KUKA KRL program: MyProgram_336().src

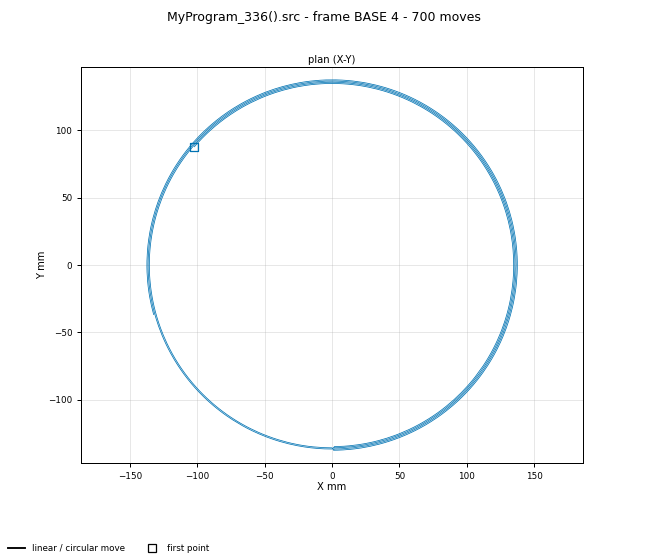
[picture p0: tool path of MyProgram_336().src in frame BASE 4, 700 of 700 moves have a stored position in this frame; points joined in program order, loops and branches not executed]
&ACCESS RVP
&REL 1
&PARAM TEMPLATE = C:\KRC\Roboter\Template\vorgabe
&PARAM EDITMASK = *
DEF MyProgram_336()
; ---- Setting reference (Base) ----
$BASE = BASE_DATA[4]

; --------------------------
; ---- Setting tool (TCP) ----
$TOOL = TOOL_DATA[3]
; --------------------------

$VEL.CP = VEL_APROX_PRINT
Startdeposition()
$VEL.CP = VEL_PRINT
LIN {X -102.3113,Y 87.8805,Z 190,A 136.75,B 1.0314,C -0.0375,E1 0.9175,E2 317.7495} C_DIS
LIN {X -99.637,Y 90.9019,Z 190,A 134.8768,B 1.0314,C -0.0407,E1 0.9211,E2 319.6393} C_DIS
LIN {X -96.5901,Y 94.1334,Z 190,A 132.7694,B 1.0312,C -0.0441,E1 0.9252,E2 321.7696} C_DIS
LIN {X -92.9272,Y 97.7507,Z 190,A 130.473,B 1.031,C -0.0478,E1 0.9299,E2 324.0767} C_DIS
LIN {X -90.6554,Y 99.8606,Z 190,A 129.0008,B 1.031,C -0.0499,E1 0.933,E2 325.565} C_DIS
LIN {X -87.4566,Y 102.6738,Z 190,A 127.0141,B 1.0308,C -0.0527,E1 0.9372,E2 327.5698} C_DIS
LIN {X -83.8464,Y 105.6426,Z 190,A 124.8651,B 1.0306,C -0.0556,E1 0.942,E2 329.7352} C_DIS
LIN {X -79.6041,Y 108.8753,Z 190,A 122.7567,B 1.0305,C -0.0588,E1 0.9467,E2 331.8252} C_DIS
LIN {X -75.5574,Y 111.7212,Z 190,A 120.2221,B 1.0303,C -0.0612,E1 0.9527,E2 334.4052} C_DIS
LIN {X -71.0559,Y 114.6372,Z 190,A 118.0805,B 1.0301,C -0.064,E1 0.9577,E2 336.5308} C_DIS
LIN {X -66.7987,Y 117.1687,Z 190,A 115.5078,B 1.0301,C -0.0659,E1 0.9641,E2 339.1524} C_DIS
LIN {X -63.7892,Y 118.8339,Z 190,A 114.076,B 1.0299,C -0.0674,E1 0.9676,E2 340.5803} C_DIS
LIN {X -60.168,Y 120.7068,Z 190,A 112.074,B 1.0299,C -0.0687,E1 0.9727,E2 342.61} C_DIS
LIN {X -55.6939,Y 122.8359,Z 190,A 110.1767,B 1.0297,C -0.0706,E1 0.9775,E2 344.4841} C_DIS
LIN {X -53.3762,Y 123.8589,Z 190,A 108.9368,B 1.0297,C -0.0712,E1 0.9808,E2 345.7408} C_DIS
LIN {X -50.0858,Y 125.2261,Z 190,A 107.31,B 1.0297,C -0.0721,E1 0.9851,E2 347.3788} C_DIS
LIN {X -46.763,Y 126.5053,Z 190,A 105.8623,B 1.0295,C -0.073,E1 0.9889,E2 348.8188} C_DIS
LIN {X -42.2008,Y 128.0989,Z 190,A 103.8391,B 1.0295,C -0.0741,E1 0.9943,E2 350.8378} C_DIS
LIN {X -39.3457,Y 129.0038,Z 190,A 102.4581,B 1.0295,C -0.0745,E1 0.998,E2 352.2297} C_DIS
LIN {X -36.135,Y 129.9398,Z 190,A 100.9752,B 1.0295,C -0.0749,E1 1.0021,E2 353.7185} C_DIS
LIN {X -32.8396,Y 130.8119,Z 190,A 99.599,B 1.0294,C -0.0754,E1 1.0058,E2 355.0863} C_DIS
LIN {X -29.9981,Y 131.4922,Z 190,A 98.2261,B 1.0294,C -0.0754,E1 1.0096,E2 356.4725} C_DIS
LIN {X -26.2178,Y 132.2996,Z 190,A 96.5812,B 1.0294,C -0.0757,E1 1.0142,E2 358.1171} C_DIS
LIN {X -20.3497,Y 133.327,Z 190,A 94.0999,B 1.0294,C -0.0759,E1 1.0211,E2 360.5919} C_DIS
LIN {X -16.2447,Y 133.8892,Z 190,A 92.3486,B 1.0294,C -0.0759,E1 1.026,E2 362.3415} C_DIS
LIN {X -12.8323,Y 134.259,Z 190,A 90.8849,B 1.0294,C -0.0756,E1 1.0301,E2 363.8052} C_DIS
LIN {X -8.2772,Y 134.6166,Z 190,A 89.0248,B 1.0294,C -0.0753,E1 1.0353,E2 365.6559} C_DIS
LIN {X -4.9946,Y 134.7786,Z 190,A 87.4221,B 1.0294,C -0.0744,E1 1.0399,E2 367.2799} C_DIS
LIN {X -0.1697,Y 134.872,Z 190,A 85.4609,B 1.0294,C -0.0738,E1 1.0454,E2 369.2309} C_DIS
LIN {X 3.9569,Y 134.813,Z 190,A 83.7686,B 1.0295,C -0.0731,E1 1.0502,E2 370.9162} C_DIS
LIN {X 8.1399,Y 134.6251,Z 190,A 82.1087,B 1.0295,C -0.0724,E1 1.0548,E2 372.5628} C_DIS
LIN {X 11.7899,Y 134.3552,Z 190,A 80.705,B 1.0296,C -0.0718,E1 1.0587,E2 373.95} C_DIS
LIN {X 15.0526,Y 134.0296,Z 190,A 79.3206,B 1.0296,C -0.0708,E1 1.0626,E2 375.333} C_DIS
LIN {X 18.9857,Y 133.5278,Z 190,A 77.6744,B 1.0298,C -0.0696,E1 1.0672,E2 376.9746} C_DIS
LIN {X 22.5244,Y 132.9769,Z 190,A 76.1298,B 1.0298,C -0.0683,E1 1.0715,E2 378.5212} C_DIS
LIN {X 26.8707,Y 132.1668,Z 190,A 74.3853,B 1.03,C -0.0669,E1 1.0763,E2 380.2509} C_DIS
LIN {X 30.9711,Y 131.268,Z 190,A 72.7965,B 1.03,C -0.0657,E1 1.0806,E2 381.8185} C_DIS
LIN {X 33.4746,Y 130.6507,Z 190,A 71.6675,B 1.0301,C -0.0645,E1 1.0837,E2 382.9507} C_DIS
LIN {X 37.5809,Y 129.5293,Z 190,A 69.9323,B 1.0302,C -0.0626,E1 1.0884,E2 384.6777} C_DIS
LIN {X 41.1171,Y 128.4501,Z 190,A 68.1111,B 1.0304,C -0.0599,E1 1.0934,E2 386.5253} C_DIS
LIN {X 44.8572,Y 127.1943,Z 190,A 66.979,B 1.0304,C -0.0596,E1 1.0963,E2 387.5987} C_DIS
LIN {X 49.4196,Y 125.4914,Z 190,A 64.9699,B 1.0306,C -0.057,E1 1.1015,E2 389.6009} C_DIS
LIN {X 52.5027,Y 124.2329,Z 190,A 63.4716,B 1.0306,C -0.0547,E1 1.1055,E2 391.108} C_DIS
LIN {X 56.3475,Y 122.5359,Z 190,A 61.913,B 1.0308,C -0.0529,E1 1.1094,E2 392.6417} C_DIS
LIN {X 59.8944,Y 120.8418,Z 190,A 60.3889,B 1.0308,C -0.0508,E1 1.1132,E2 394.1497} C_DIS
LIN {X 65.5035,Y 117.8978,Z 190,A 58.0418,B 1.031,C -0.0478,E1 1.119,E2 396.4588} C_DIS
LIN {X 68.3222,Y 116.2869,Z 190,A 56.6628,B 1.0311,C -0.0454,E1 1.1223,E2 397.8377} C_DIS
LIN {X 71.8669,Y 114.1303,Z 190,A 54.9703,B 1.0313,C -0.0426,E1 1.1263,E2 399.5224} C_DIS
LIN {X 74.5809,Y 112.376,Z 190,A 53.7411,B 1.0313,C -0.0407,E1 1.1292,E2 400.7356} C_DIS
LIN {X 78.1084,Y 109.9537,Z 190,A 52.01,B 1.0314,C -0.0377,E1 1.1332,E2 402.4571} C_DIS
LIN {X 81.7669,Y 107.2603,Z 190,A 50.3364,B 1.0315,C -0.035,E1 1.1369,E2 404.102} C_DIS
LIN {X 84.8066,Y 104.8734,Z 190,A 48.8019,B 1.0316,C -0.0322,E1 1.1402,E2 405.6245} C_DIS
LIN {X 88.0931,Y 102.1282,Z 190,A 47.1444,B 1.0317,C -0.0292,E1 1.1437,E2 407.264} C_DIS
LIN {X 91.5195,Y 99.0698,Z 190,A 45.3771,B 1.0318,C -0.0259,E1 1.1473,E2 409.0107} C_DIS
LIN {X 93.7332,Y 96.9776,Z 190,A 44.1924,B 1.0318,C -0.0236,E1 1.1497,E2 410.1831} C_DIS
LIN {X 96.9928,Y 93.7175,Z 190,A 42.4386,B 1.0319,C -0.0203,E1 1.1531,E2 411.9139} C_DIS
LIN {X 99.9264,Y 90.583,Z 190,A 40.7946,B 1.0319,C -0.017,E1 1.1562,E2 413.5376} C_DIS
LIN {X 102.9019,Y 87.1883,Z 190,A 39.069,B 1.032,C -0.0135,E1 1.1593,E2 415.2415} C_DIS
LIN {X 105.5381,Y 83.9777,Z 190,A 37.4765,B 1.032,C -0.0102,E1 1.1621,E2 416.8145} C_DIS
LIN {X 108.1139,Y 80.6346,Z 190,A 36.0003,B 1.0321,C -0.0075,E1 1.1646,E2 418.2544} C_DIS
LIN {X 110.3862,Y 77.4954,Z 190,A 34.2134,B 1.0321,C -0.0029,E1 1.1675,E2 420.0579} C_DIS
LIN {X 112.2299,Y 74.7998,Z 190,A 33.1847,B 1.0321,C -0.0012,E1 1.169,E2 421.0454} C_DIS
LIN {X 114.6113,Y 71.0975,Z 190,A 31.5626,B 1.0321,C 0.0022,E1 1.1714,E2 422.6389} C_DIS
LIN {X 116.9008,Y 67.2672,Z 190,A 29.7748,B 1.0321,C 0.0065,E1 1.1739,E2 424.4146} C_DIS
LIN {X 118.7485,Y 63.9481,Z 190,A 28.4203,B 1.0321,C 0.0093,E1 1.1757,E2 425.739} C_DIS
LIN {X 120.388,Y 60.8022,Z 190,A 27.1011,B 1.0321,C 0.0122,E1 1.1774,E2 427.0364} C_DIS
LIN {X 122.4869,Y 56.4534,Z 190,A 25.2811,B 1.0321,C 0.0164,E1 1.1795,E2 428.8296} C_DIS
LIN {X 124.0395,Y 52.9585,Z 190,A 23.9004,B 1.0319,C 0.0194,E1 1.181,E2 430.1818} C_DIS
LIN {X 125.287,Y 49.9347,Z 190,A 22.621,B 1.0319,C 0.0225,E1 1.1824,E2 431.4484} C_DIS
LIN {X 126.9081,Y 45.6549,Z 190,A 20.9084,B 1.0318,C 0.0265,E1 1.184,E2 433.1339} C_DIS
LIN {X 127.9726,Y 42.58,Z 190,A 19.6934,B 1.0318,C 0.0294,E1 1.1851,E2 434.3292} C_DIS
LIN {X 129.125,Y 38.9496,Z 190,A 18.2521,B 1.0316,C 0.0328,E1 1.1863,E2 435.7498} C_DIS
LIN {X 130.0995,Y 35.5641,Z 190,A 16.9404,B 1.0316,C 0.0359,E1 1.1872,E2 437.0398} C_DIS
LIN {X 130.8248,Y 32.7889,Z 190,A 15.8845,B 1.0314,C 0.0384,E1 1.188,E2 438.0763} C_DIS
LIN {X 131.5462,Y 29.7614,Z 190,A 14.7035,B 1.0314,C 0.0413,E1 1.1887,E2 439.2406} C_DIS
LIN {X 132.2329,Y 26.5457,Z 190,A 13.4674,B 1.0312,C 0.0443,E1 1.1894,E2 440.4576} C_DIS
LIN {X 132.8388,Y 23.327,Z 190,A 12.2792,B 1.0311,C 0.0471,E1 1.19,E2 441.6216} C_DIS
LIN {X 133.4079,Y 19.8242,Z 190,A 10.9318,B 1.0309,C 0.0504,E1 1.1905,E2 442.95} C_DIS
LIN {X 133.8223,Y 16.7998,Z 190,A 9.5869,B 1.0307,C 0.0543,E1 1.191,E2 444.3014} C_DIS
LIN {X 134.3804,Y 11.4921,Z 190,A 7.7327,B 1.0305,C 0.0584,E1 1.1915,E2 446.1055} C_DIS
LIN {X 134.6681,Y 7.4209,Z 190,A 6.3001,B 1.0303,C 0.0616,E1 1.1918,E2 447.5015} C_DIS
LIN {X 134.7793,Y 4.9766,Z 190,A 5.324,B 1.0301,C 0.0642,E1 1.1918,E2 448.4702} C_DIS
LIN {X 134.8718,Y 0.2243,Z 190,A 3.6075,B 1.0299,C 0.0682,E1 1.1919,E2 450.1498} C_DIS
LIN {X 134.8428,Y -2.814,Z 190,A 2.2229,B 1.0296,C 0.0723,E1 1.1919,E2 451.5469} C_DIS
LIN {X 134.6641,Y -7.5005,Z 190,A 0.6838,B 1.0294,C 0.0754,E1 1.1917,E2 453.03} C_DIS
LIN {X 134.3382,Y -11.9912,Z 190,A -1.3076,B 1.0289,C 0.0812,E1 1.1912,E2 455.0324} C_DIS
LIN {X 133.9962,Y -15.3478,Z 190,A -2.2241,B 1.0289,C 0.0824,E1 1.191,E2 455.8842} C_DIS
LIN {X 133.6072,Y -18.4298,Z 190,A -3.5585,B 1.0285,C 0.0861,E1 1.1905,E2 457.2212} C_DIS
LIN {X 132.9067,Y -22.945,Z 190,A -5.1491,B 1.0282,C 0.0896,E1 1.1898,E2 458.7683} C_DIS
LIN {X 132.425,Y -25.5689,Z 190,A -6.1171,B 1.028,C 0.0918,E1 1.1893,E2 459.7157} C_DIS
LIN {X 131.6541,Y -29.2892,Z 190,A -7.6683,B 1.0277,C 0.0959,E1 1.1884,E2 461.2599} C_DIS
LIN {X 130.7208,Y -33.1985,Z 190,A -9.1638,B 1.0273,C 0.0995,E1 1.1874,E2 462.7291} C_DIS
LIN {X 129.6374,Y -37.2116,Z 190,A -11.2094,B 1.0267,C 0.1058,E1 1.1858,E2 464.812} C_DIS
LIN {X 128.1582,Y -42.0227,Z 190,A -12.4751,B 1.0266,C 0.1069,E1 1.1848,E2 465.966} C_DIS
LIN {X 127.2027,Y -44.833,Z 190,A -13.6596,B 1.0263,C 0.1098,E1 1.1838,E2 467.1414} C_DIS
LIN {X 126.0621,Y -47.9462,Z 190,A -14.8848,B 1.026,C 0.1126,E1 1.1826,E2 468.3436} C_DIS
LIN {X 124.9341,Y -50.81,Z 190,A -16.3072,B 1.0255,C 0.1166,E1 1.1811,E2 469.7819} C_DIS
LIN {X 122.8544,Y -55.6527,Z 190,A -18.0514,B 1.0251,C 0.1199,E1 1.1792,E2 471.4627} C_DIS
LIN {X 121.7034,Y -58.1231,Z 190,A -19.1462,B 1.0248,C 0.1225,E1 1.1779,E2 472.5499} C_DIS
LIN {X 119.7934,Y -61.9695,Z 190,A -20.702,B 1.0244,C 0.1258,E1 1.176,E2 474.0716} C_DIS
LIN {X 118.0054,Y -65.3091,Z 190,A -22.1982,B 1.024,C 0.1293,E1 1.174,E2 475.5539} C_DIS
LIN {X 115.8653,Y -69.0347,Z 190,A -23.7083,B 1.0236,C 0.1322,E1 1.1719,E2 477.0234} C_DIS
LIN {X 113.9593,Y -72.1378,Z 190,A -25.1095,B 1.0232,C 0.1353,E1 1.1699,E2 478.4062} C_DIS
LIN {X 112.1061,Y -74.9853,Z 190,A -26.594,B 1.0227,C 0.139,E1 1.1676,E2 479.8974} C_DIS
LIN {X 106.1881,Y -83.1545,Z 190,A -30.2178,B 1.0218,C 0.1459,E1 1.1617,E2 483.4355} C_DIS
LIN {X 104.0205,Y -85.8506,Z 190,A -32.1493,B 1.0209,C 0.1516,E1 1.1582,E2 485.4304} C_DIS
LIN {X 100.756,Y -89.6603,Z 190,A -33.3836,B 1.0209,C 0.1519,E1 1.1561,E2 486.5452} C_DIS
LIN {X 95.9069,Y -94.8289,Z 190,A -36.3467,B 1.0199,C 0.1583,E1 1.1504,E2 489.5043} C_DIS
LIN {X 90.6268,Y -99.8866,Z 190,A -38.942,B 1.0193,C 0.1624,E1 1.1452,E2 492.0322} C_DIS
LIN {X 84.6508,Y -104.999,Z 190,A -42.6037,B 1.0179,C 0.1707,E1 1.1373,E2 495.7404} C_DIS
LIN {X 80.9291,Y -107.894,Z 190,A -43.8915,B 1.0179,C 0.1712,E1 1.1346,E2 496.9318} C_DIS
LIN {X 78.2121,Y -109.8795,Z 190,A -45.324,B 1.0174,C 0.1739,E1 1.1313,E2 498.3657} C_DIS
LIN {X 74.889,Y -112.1704,Z 190,A -46.9282,B 1.0169,C 0.1766,E1 1.1276,E2 499.956} C_DIS
LIN {X 71.4377,Y -114.3995,Z 190,A -48.5106,B 1.0165,C 0.1789,E1 1.1239,E2 501.5172} C_DIS
LIN {X 66.7848,Y -117.1765,Z 190,A -50.4352,B 1.0161,C 0.1812,E1 1.1194,E2 503.3913} C_DIS
LIN {X 64.1989,Y -118.6138,Z 190,A -51.8491,B 1.0156,C 0.1839,E1 1.1158,E2 504.8279} C_DIS
LIN {X 60.9277,Y -120.3242,Z 190,A -53.1719,B 1.0154,C 0.1854,E1 1.1126,E2 506.1177} C_DIS
LIN {X 57.1495,Y -122.1651,Z 190,A -54.7355,B 1.015,C 0.1872,E1 1.1087,E2 507.6517} C_DIS
LIN {X 50.0805,Y -125.2282,Z 190,A -57.8745,B 1.0142,C 0.1913,E1 1.1006,E2 510.7745} C_DIS
LIN {X 46.6988,Y -126.5294,Z 190,A -59.694,B 1.0136,C 0.1945,E1 1.0957,E2 512.6342} C_DIS
LIN {X 43.1235,Y -127.7916,Z 190,A -60.7374,B 1.0136,C 0.1943,E1 1.0931,E2 513.5994} C_DIS
LIN {X 40.4042,Y -128.6779,Z 190,A -61.97,B 1.0134,C 0.1958,E1 1.0898,E2 514.8354} C_DIS
LIN {X 37.734,Y -129.4845,Z 190,A -63.1158,B 1.0131,C 0.1971,E1 1.0867,E2 515.9765} C_DIS
LIN {X 34.6217,Y -130.3511,Z 190,A -64.3488,B 1.013,C 0.1981,E1 1.0834,E2 517.1907} C_DIS
LIN {X 31.3438,Y -131.1782,Z 190,A -65.8293,B 1.0126,C 0.1997,E1 1.0793,E2 518.6785} C_DIS
LIN {X 27.9921,Y -131.9347,Z 190,A -67.1371,B 1.0124,C 0.2006,E1 1.0758,E2 519.9659} C_DIS
LIN {X 24.3157,Y -132.6618,Z 190,A -68.7166,B 1.0122,C 0.2021,E1 1.0714,E2 521.5447} C_DIS
LIN {X 19.7753,Y -133.4139,Z 190,A -71.0449,B 1.0116,C 0.205,E1 1.0648,E2 523.9265} C_DIS
LIN {X 15.397,Y -133.9903,Z 190,A -72.2873,B 1.0117,C 0.2043,E1 1.0615,E2 525.0811} C_DIS
LIN {X 12.6782,Y -134.2738,Z 190,A -73.5571,B 1.0115,C 0.2054,E1 1.0579,E2 526.3668} C_DIS
LIN {X 8.7907,Y -134.585,Z 190,A -75.5639,B 1.011,C 0.2076,E1 1.0521,E2 528.4237} C_DIS
LIN {X 4.4935,Y -134.7977,Z 190,A -76.8327,B 1.0112,C 0.2068,E1 1.0488,E2 529.615} C_DIS
LIN {X 1.7112,Y -134.8611,Z 190,A -78.397,B 1.0108,C 0.2085,E1 1.0442,E2 531.2338} C_DIS
LIN {X 1.7112,Y -134.8611,Z 190,A -78.397,B 1.0108,C 0.2085,E1 1.0442,E2 531.2338} C_DIS
Enddeposition()
LIN {X 0.9737,Y -135.7663,Z 190,A -78.1161,B 1.011,C 0.2073,E1 1.045,E2 530.8941} C_DIS
Startdeposition()
$VEL.CP = VEL_PRINT
LIN {X 6.9745,Y -135.5906,Z 190,A -75.108,B 1.0116,C 0.2046,E1 1.0537,E2 527.8168} C_DIS
LIN {X 15.8798,Y -134.8379,Z 190,A -71.5086,B 1.012,C 0.2026,E1 1.0638,E2 524.2401} C_DIS
LIN {X 22.5103,Y -133.8906,Z 190,A -68.8862,B 1.0123,C 0.2009,E1 1.071,E2 521.6453} C_DIS
LIN {X 25.8344,Y -133.2894,Z 190,A -67.4107,B 1.0126,C 0.1994,E1 1.0751,E2 520.1618} C_DIS
LIN {X 28.9884,Y -132.6392,Z 190,A -66.1615,B 1.0128,C 0.1985,E1 1.0785,E2 518.9274} C_DIS
LIN {X 33.1343,Y -131.6645,Z 190,A -64.4396,B 1.0131,C 0.1969,E1 1.0832,E2 517.2151} C_DIS
LIN {X 36.5609,Y -130.7541,Z 190,A -63.091,B 1.0133,C 0.1958,E1 1.0869,E2 515.8865} C_DIS
LIN {X 39.6778,Y -129.8422,Z 190,A -61.7393,B 1.0136,C 0.1943,E1 1.0905,E2 514.5366} C_DIS
LIN {X 42.6723,Y -128.8893,Z 190,A -60.4442,B 1.0139,C 0.1928,E1 1.094,E2 513.245} C_DIS
LIN {X 47.1805,Y -127.3088,Z 190,A -58.7448,B 1.0141,C 0.1914,E1 1.0984,E2 511.5893} C_DIS
LIN {X 49.6539,Y -126.3647,Z 190,A -56.71,B 1.0151,C 0.1861,E1 1.1041,E2 509.4227} C_DIS
LIN {X 55.9848,Y -123.6906,Z 190,A -54.8821,B 1.0151,C 0.1864,E1 1.1084,E2 507.7458} C_DIS
LIN {X 59.6108,Y -121.984,Z 190,A -53.2483,B 1.0155,C 0.184,E1 1.1125,E2 506.1189} C_DIS
LIN {X 62.986,Y -120.2749,Z 190,A -51.8669,B 1.0158,C 0.1824,E1 1.1159,E2 504.7667} C_DIS
LIN {X 66.363,Y -118.4475,Z 190,A -49.6176,B 1.0167,C 0.177,E1 1.1216,E2 502.4272} C_DIS
LIN {X 71.4623,Y -115.4429,Z 190,A -47.9158,B 1.0169,C 0.1762,E1 1.1254,E2 500.8363} C_DIS
LIN {X 74.8801,Y -113.2558,Z 190,A -46.4071,B 1.0173,C 0.1741,E1 1.1289,E2 499.3549} C_DIS
LIN {X 77.3617,Y -111.5753,Z 190,A -45.1498,B 1.0176,C 0.1718,E1 1.1318,E2 498.0977} C_DIS
LIN {X 82.7712,Y -107.6238,Z 190,A -42.5903,B 1.0183,C 0.1676,E1 1.1375,E2 495.5736} C_DIS
LIN {X 86.0264,Y -105.0396,Z 190,A -40.5384,B 1.0191,C 0.1627,E1 1.1421,E2 493.4787} C_DIS
LIN {X 89.8971,Y -101.7465,Z 190,A -38.9851,B 1.0194,C 0.1611,E1 1.1452,E2 492.0065} C_DIS
LIN {X 93.6072,Y -98.3443,Z 190,A -37.1127,B 1.0199,C 0.1579,E1 1.149,E2 490.1675} C_DIS
LIN {X 96.9051,Y -95.0959,Z 190,A -34.9295,B 1.0207,C 0.1525,E1 1.1533,E2 487.9509} C_DIS
LIN {X 100.2823,Y -91.5282,Z 190,A -33.4715,B 1.0209,C 0.151,E1 1.1559,E2 486.5768} C_DIS
LIN {X 104.4413,Y -86.7519,Z 190,A -31.0792,B 1.0216,C 0.1463,E1 1.1602,E2 484.2211} C_DIS
LIN {X 109.0323,Y -80.9064,Z 190,A -28.199,B 1.0225,C 0.1403,E1 1.1651,E2 481.3739} C_DIS
LIN {X 113.3577,Y -74.7254,Z 190,A -25.4327,B 1.0232,C 0.1347,E1 1.1694,E2 478.6624} C_DIS
LIN {X 115.8481,Y -70.8032,Z 190,A -23.9195,B 1.0235,C 0.1322,E1 1.1716,E2 477.2086} C_DIS
LIN {X 117.5871,Y -67.8759,Z 190,A -22.4205,B 1.024,C 0.1283,E1 1.1737,E2 475.7001} C_DIS
LIN {X 119.8326,Y -63.8285,Z 190,A -20.645,B 1.0245,C 0.1243,E1 1.176,E2 473.9472} C_DIS
LIN {X 121.6063,Y -60.3763,Z 190,A -19.3533,B 1.0248,C 0.1219,E1 1.1776,E2 472.7009} C_DIS
LIN {X 123.017,Y -57.4489,Z 190,A -18.0289,B 1.0252,C 0.1186,E1 1.1792,E2 471.3818} C_DIS
LIN {X 124.5269,Y -54.0963,Z 190,A -16.0232,B 1.0259,C 0.1121,E1 1.1815,E2 469.3139} C_DIS
LIN {X 126.7317,Y -48.7098,Z 190,A -14.4966,B 1.0261,C 0.1106,E1 1.1829,E2 467.9106} C_DIS
LIN {X 129.6888,Y -40.179,Z 190,A -11.0276,B 1.027,C 0.1023,E1 1.186,E2 464.4846} C_DIS
LIN {X 130.8301,Y -36.2891,Z 190,A -9.5625,B 1.0273,C 0.0989,E1 1.1871,E2 463.0508} C_DIS
LIN {X 131.8524,Y -32.3826,Z 190,A -8.0428,B 1.0276,C 0.0953,E1 1.1881,E2 461.5544} C_DIS
LIN {X 132.804,Y -28.225,Z 190,A -6.4515,B 1.028,C 0.0915,E1 1.1891,E2 459.9894} C_DIS
LIN {X 133.632,Y -23.9971,Z 190,A -4.9377,B 1.0283,C 0.0881,E1 1.1898,E2 458.5143} C_DIS
LIN {X 134.1433,Y -20.952,Z 190,A -3.7879,B 1.0285,C 0.0854,E1 1.1903,E2 457.3836} C_DIS
LIN {X 134.6414,Y -17.4673,Z 190,A -1.6977,B 1.0291,C 0.0779,E1 1.1911,E2 455.2133} C_DIS
LIN {X 135.3223,Y -11.0204,Z 190,A 0.051,B 1.0293,C 0.0757,E1 1.1915,E2 453.5921} C_DIS
LIN {X 135.5533,Y -7.6919,Z 190,A 1.7384,B 1.0296,C 0.0703,E1 1.1918,E2 451.8677} C_DIS
LIN {X 135.745,Y -2.6227,Z 190,A 3.0238,B 1.0297,C 0.0689,E1 1.1918,E2 450.6915} C_DIS
LIN {X 135.7107,Y 4.0127,Z 190,A 5.6323,B 1.0302,C 0.0622,E1 1.1918,E2 448.1062} C_DIS
LIN {X 135.4983,Y 8.5847,Z 190,A 7.7512,B 1.0305,C 0.0557,E1 1.1914,E2 445.9623} C_DIS
LIN {X 135.0989,Y 13.4892,Z 190,A 9.3749,B 1.0307,C 0.0524,E1 1.191,E2 444.3954} C_DIS
LIN {X 134.6912,Y 17.0876,Z 190,A 10.5353,B 1.0308,C 0.0501,E1 1.1906,E2 443.2809} C_DIS
LIN {X 134.0881,Y 21.3087,Z 190,A 11.9098,B 1.0309,C 0.0474,E1 1.19,E2 441.9589} C_DIS
LIN {X 133.4862,Y 24.805,Z 190,A 13.3118,B 1.0311,C 0.0438,E1 1.1893,E2 440.5682} C_DIS
LIN {X 132.8466,Y 28.0274,Z 190,A 14.6057,B 1.0312,C 0.0405,E1 1.1886,E2 439.2852} C_DIS
LIN {X 131.9947,Y 31.7922,Z 190,A 15.9489,B 1.0314,C 0.0375,E1 1.1878,E2 437.9768} C_DIS
LIN {X 131.3208,Y 34.4742,Z 190,A 17.0801,B 1.0314,C 0.0345,E1 1.187,E2 436.8497} C_DIS
LIN {X 130.3166,Y 38.0909,Z 190,A 18.4506,B 1.0316,C 0.0313,E1 1.186,E2 435.5049} C_DIS
LIN {X 129.0944,Y 42.0543,Z 190,A 20.0951,B 1.0316,C 0.0272,E1 1.1846,E2 433.8729} C_DIS
LIN {X 127.6763,Y 46.1746,Z 190,A 22.1395,B 1.0318,C 0.0212,E1 1.1826,E2 431.8025} C_DIS
LIN {X 125.8411,Y 50.9644,Z 190,A 23.4871,B 1.0318,C 0.0197,E1 1.1813,E2 430.5545} C_DIS
LIN {X 124.4351,Y 54.3084,Z 190,A 25.3938,B 1.0319,C 0.0137,E1 1.1792,E2 428.6014} C_DIS
LIN {X 122.3616,Y 58.8305,Z 190,A 26.73,B 1.0319,C 0.0121,E1 1.1777,E2 427.3577} C_DIS
LIN {X 120.5356,Y 62.4896,Z 190,A 28.2924,B 1.0319,C 0.0085,E1 1.1757,E2 425.8145} C_DIS
LIN {X 118.5328,Y 66.2113,Z 190,A 29.8531,B 1.032,C 0.0051,E1 1.1736,E2 424.2802} C_DIS
LIN {X 115.3809,Y 71.5621,Z 190,A 32.0788,B 1.032,C 0.0005,E1 1.1705,E2 422.1011} C_DIS
LIN {X 111.8105,Y 77.0214,Z 190,A 34.7055,B 1.032,C -0.0056,E1 1.1665,E2 419.489} C_DIS
LIN {X 109.234,Y 80.6341,Z 190,A 36.3939,B 1.032,C -0.0092,E1 1.1637,E2 417.8221} C_DIS
LIN {X 106.6472,Y 84.0252,Z 190,A 37.9571,B 1.032,C -0.0123,E1 1.1611,E2 416.2865} C_DIS
LIN {X 103.9872,Y 87.2954,Z 190,A 39.5647,B 1.032,C -0.0156,E1 1.1583,E2 414.6988} C_DIS
LIN {X 101.2428,Y 90.4641,Z 190,A 41.1743,B 1.0319,C -0.0189,E1 1.1553,E2 413.1077} C_DIS
LIN {X 98.3318,Y 93.6203,Z 190,A 42.8372,B 1.0318,C -0.0223,E1 1.1522,E2 411.462} C_DIS
LIN {X 95.2112,Y 96.792,Z 190,A 44.5361,B 1.0318,C -0.0255,E1 1.1488,E2 409.7836} C_DIS
LIN {X 92.4492,Y 99.4333,Z 190,A 45.9579,B 1.0317,C -0.0281,E1 1.146,E2 408.3839} C_DIS
LIN {X 89.1391,Y 102.4113,Z 190,A 47.6486,B 1.0316,C -0.0312,E1 1.1425,E2 406.7149} C_DIS
LIN {X 85.8965,Y 105.1457,Z 190,A 49.2862,B 1.0315,C -0.0341,E1 1.1389,E2 405.0947} C_DIS
LIN {X 82.7379,Y 107.6493,Z 190,A 50.8896,B 1.0314,C -0.037,E1 1.1354,E2 403.5025} C_DIS
LIN {X 79.2771,Y 110.223,Z 190,A 52.5654,B 1.0313,C -0.0399,E1 1.1317,E2 401.8432} C_DIS
LIN {X 75.5839,Y 112.7872,Z 190,A 54.1264,B 1.0312,C -0.042,E1 1.1281,E2 400.3205} C_DIS
LIN {X 70.6551,Y 115.939,Z 190,A 57.3158,B 1.0309,C -0.0492,E1 1.1203,E2 397.0491} C_DIS
LIN {X 64.888,Y 119.2619,Z 190,A 59.1439,B 1.0309,C -0.0501,E1 1.1161,E2 395.3328} C_DIS
LIN {X 61.4972,Y 121.0429,Z 190,A 60.5279,B 1.0307,C -0.0518,E1 1.1127,E2 393.975} C_DIS
LIN {X 58.33,Y 122.6007,Z 190,A 61.9379,B 1.0307,C -0.0538,E1 1.1091,E2 392.5741} C_DIS
LIN {X 55.5064,Y 123.9045,Z 190,A 63.5523,B 1.0305,C -0.0568,E1 1.1049,E2 390.9261} C_DIS
LIN {X 51.7728,Y 125.5119,Z 190,A 64.8855,B 1.0305,C -0.0579,E1 1.1015,E2 389.6361} C_DIS
LIN {X 44.4676,Y 128.2807,Z 190,A 67.8948,B 1.0302,C -0.0612,E1 1.0937,E2 386.6593} C_DIS
LIN {X 40.2663,Y 129.6621,Z 190,A 69.6034,B 1.0302,C -0.063,E1 1.0891,E2 384.9686} C_DIS
LIN {X 36.819,Y 130.6819,Z 190,A 71.0445,B 1.03,C -0.0645,E1 1.0852,E2 383.5361} C_DIS
LIN {X 33.6111,Y 131.5435,Z 190,A 72.3201,B 1.03,C -0.0656,E1 1.0818,E2 382.2748} C_DIS
LIN {X 30.4634,Y 132.3079,Z 190,A 73.7168,B 1.0298,C -0.0671,E1 1.0779,E2 380.8752} C_DIS
LIN {X 27.0172,Y 133.0543,Z 190,A 75.0998,B 1.0298,C -0.0682,E1 1.0742,E2 379.5041} C_DIS
LIN {X 23.4779,Y 133.7249,Z 190,A 76.5996,B 1.0297,C -0.0695,E1 1.07,E2 378.007} C_DIS
LIN {X 18.5954,Y 134.4916,Z 190,A 78.5273,B 1.0297,C -0.0708,E1 1.0647,E2 376.0972} C_DIS
LIN {X 15.3082,Y 134.9056,Z 190,A 79.8861,B 1.0295,C -0.0717,E1 1.0609,E2 374.7432} C_DIS
LIN {X 12.009,Y 135.2388,Z 190,A 81.1532,B 1.0295,C -0.0723,E1 1.0573,E2 373.4909} C_DIS
LIN {X 7.9358,Y 135.5382,Z 190,A 83.4145,B 1.0293,C -0.0748,E1 1.0508,E2 371.1714} C_DIS
LIN {X 3.6061,Y 135.722,Z 190,A 84.8053,B 1.0293,C -0.0746,E1 1.047,E2 369.8292} C_DIS
LIN {X 0.0822,Y 135.7715,Z 190,A 86.7533,B 1.0293,C -0.0763,E1 1.0414,E2 367.8315} C_DIS
LIN {X -4.7567,Y 135.6875,Z 190,A 88.1933,B 1.0293,C -0.0756,E1 1.0375,E2 366.4581} C_DIS
LIN {X -11.4564,Y 135.2855,Z 190,A 91.0152,B 1.0293,C -0.0763,E1 1.0295,E2 363.6385} C_DIS
LIN {X -15.8046,Y 134.8469,Z 190,A 92.5828,B 1.0293,C -0.0759,E1 1.0252,E2 362.1016} C_DIS
LIN {X -18.0914,Y 134.5597,Z 190,A 93.9839,B 1.0292,C -0.0769,E1 1.0212,E2 360.6546} C_DIS
LIN {X -23.5002,Y 133.721,Z 190,A 96.1359,B 1.0292,C -0.0765,E1 1.0152,E2 358.5208} C_DIS
LIN {X -26.5632,Y 133.1467,Z 190,A 97.4694,B 1.0292,C -0.0764,E1 1.0115,E2 357.1858} C_DIS
LIN {X -29.7492,Y 132.4711,Z 190,A 98.8895,B 1.0292,C -0.0762,E1 1.0076,E2 355.7616} C_DIS
LIN {X -33.4098,Y 131.5946,Z 190,A 100.3858,B 1.0292,C -0.0757,E1 1.0035,E2 354.2759} C_DIS
LIN {X -36.3408,Y 130.8157,Z 190,A 101.7875,B 1.0292,C -0.0754,E1 0.9996,E2 352.8616} C_DIS
LIN {X -40.5835,Y 129.5642,Z 190,A 103.6718,B 1.0293,C -0.0747,E1 0.9946,E2 350.9765} C_DIS
LIN {X -47.0654,Y 127.3519,Z 190,A 106.6561,B 1.0294,C -0.0733,E1 0.9866,E2 347.9835} C_DIS
LIN {X -50.4976,Y 126.0293,Z 190,A 108.2694,B 1.0294,C -0.0724,E1 0.9823,E2 346.3643} C_DIS
LIN {X -53.8892,Y 124.6164,Z 190,A 109.6394,B 1.0296,C -0.0711,E1 0.9788,E2 345.0147} C_DIS
LIN {X -56.7168,Y 123.3555,Z 190,A 111.3183,B 1.0296,C -0.0705,E1 0.9744,E2 343.2961} C_DIS
LIN {X -61.2171,Y 121.1855,Z 190,A 113.4176,B 1.0297,C -0.0687,E1 0.9691,E2 341.199} C_DIS
LIN {X -64.9741,Y 119.2149,Z 190,A 115.8514,B 1.0298,C -0.0675,E1 0.9629,E2 338.6955} C_DIS
LIN {X -69.1628,Y 116.8354,Z 190,A 118.1556,B 1.03,C -0.0655,E1 0.9572,E2 336.3623} C_DIS
LIN {X -73.8523,Y 113.9284,Z 190,A 119.9156,B 1.0301,C -0.0624,E1 0.9532,E2 334.6666} C_DIS
LIN {X -77.3242,Y 111.6014,Z 190,A 121.851,B 1.0303,C -0.0602,E1 0.9486,E2 332.7134} C_DIS
LIN {X -83.9875,Y 106.6769,Z 190,A 125.5899,B 1.0305,C -0.0555,E1 0.9402,E2 328.9499} C_DIS
LIN {X -87.5679,Y 103.7586,Z 190,A 127.7382,B 1.0307,C -0.0527,E1 0.9354,E2 326.7806} C_DIS
LIN {X -90.5287,Y 101.1849,Z 190,A 129.7005,B 1.0308,C -0.0501,E1 0.9312,E2 324.785} C_DIS
LIN {X -96.1808,Y 95.8286,Z 190,A 133.1129,B 1.0311,C -0.0445,E1 0.9243,E2 321.3606} C_DIS
LIN {X -99.3804,Y 92.506,Z 190,A 135.8003,B 1.0312,C -0.041,E1 0.919,E2 318.5903} C_DIS
LIN {X -102.6438,Y 88.8717,Z 190,A 137.8153,B 1.0314,C -0.0371,E1 0.9153,E2 316.582} C_DIS
LIN {X -104.9677,Y 86.1143,Z 190,A 139.2013,B 1.0314,C -0.0341,E1 0.9128,E2 315.2124} C_DIS
LIN {X -107.4136,Y 83.0432,Z 190,A 140.9607,B 1.0316,C -0.0308,E1 0.9098,E2 313.4424} C_DIS
LIN {X -109.9941,Y 79.5936,Z 190,A 143.0721,B 1.0316,C -0.0269,E1 0.9062,E2 311.2985} C_DIS
LIN {X -112.3529,Y 76.2278,Z 190,A 145.053,B 1.0318,C -0.0231,E1 0.903,E2 309.2903} C_DIS
LIN {X -114.9299,Y 72.2841,Z 190,A 147.2603,B 1.0318,C -0.0186,E1 0.8996,E2 307.059} C_DIS
LIN {X -117.8131,Y 67.4831,Z 190,A 149.9561,B 1.032,C -0.0131,E1 0.8957,E2 304.326} C_DIS
LIN {X -119.871,Y 63.7552,Z 190,A 152.0935,B 1.032,C -0.0087,E1 0.8928,E2 302.1498} C_DIS
LIN {X -121.8048,Y 59.9741,Z 190,A 153.9118,B 1.032,C -0.0043,E1 0.8906,E2 300.3295} C_DIS
LIN {X -123.1735,Y 57.1104,Z 190,A 155.4272,B 1.032,C -0.001,E1 0.8887,E2 298.7943} C_DIS
LIN {X -124.8588,Y 53.3286,Z 190,A 157.5217,B 1.032,C 0.0036,E1 0.8863,E2 296.6598} C_DIS
LIN {X -126.4539,Y 49.4244,Z 190,A 159.4038,B 1.032,C 0.0082,E1 0.8844,E2 294.7666} C_DIS
LIN {X -127.6835,Y 46.1545,Z 190,A 161.1576,B 1.032,C 0.0122,E1 0.8826,E2 292.9804} C_DIS
LIN {X -128.6613,Y 43.3568,Z 190,A 162.6772,B 1.032,C 0.0156,E1 0.8812,E2 291.4292} C_DIS
LIN {X -129.8685,Y 39.592,Z 190,A 164.4584,B 1.0318,C 0.0201,E1 0.8797,E2 289.6355} C_DIS
LIN {X -130.8604,Y 36.1808,Z 190,A 166.3461,B 1.0318,C 0.0244,E1 0.8783,E2 287.7017} C_DIS
LIN {X -131.7574,Y 32.7682,Z 190,A 168.3205,B 1.0316,C 0.0288,E1 0.8769,E2 285.6689} C_DIS
LIN {X -132.5095,Y 29.5812,Z 190,A 169.7325,B 1.0316,C 0.0325,E1 0.876,E2 284.2541} C_DIS
LIN {X -133.3329,Y 25.607,Z 190,A 171.4827,B 1.0314,C 0.0372,E1 0.8751,E2 282.5003} C_DIS
LIN {X -133.9091,Y 22.3996,Z 190,A 173.2007,B 1.0312,C 0.0413,E1 0.8742,E2 280.7409} C_DIS
LIN {X -134.5296,Y 18.3211,Z 190,A 175.2707,B 1.031,C 0.0464,E1 0.8734,E2 278.6312} C_DIS
LIN {X -134.9718,Y 14.6987,Z 190,A 176.9373,B 1.0308,C 0.0508,E1 0.8728,E2 276.9496} C_DIS
LIN {X -135.2961,Y 11.3308,Z 190,A 178.6727,B 1.0306,C 0.055,E1 0.8724,E2 275.1766} C_DIS
LIN {X -135.5648,Y 7.4871,Z 190,A -179.36,B 1.0303,C 0.0598,E1 0.8721,E2 273.1674} C_DIS
LIN {X -135.7111,Y 3.9966,Z 190,A -177.6997,B 1.03,C 0.0641,E1 0.8719,E2 271.4844} C_DIS
LIN {X -135.7706,Y -0.2411,Z 190,A -175.6209,B 1.0297,C 0.0694,E1 0.8719,E2 269.3698} C_DIS
LIN {X -135.7166,Y -3.8,Z 190,A -173.9237,B 1.0294,C 0.0737,E1 0.8719,E2 267.6485} C_DIS
LIN {X -135.5387,Y -7.9278,Z 190,A -171.9359,B 1.029,C 0.0788,E1 0.8722,E2 265.6304} C_DIS
LIN {X -135.2894,Y -11.4096,Z 190,A -170.1193,B 1.0287,C 0.0832,E1 0.8726,E2 263.7703} C_DIS
LIN {X -134.8287,Y -15.9574,Z 190,A -168.0112,B 1.0282,C 0.0887,E1 0.8733,E2 261.6401} C_DIS
LIN {X -134.3856,Y -19.3371,Z 190,A -166.212,B 1.0278,C 0.0929,E1 0.874,E2 259.7948} C_DIS
LIN {X -133.7066,Y -23.5805,Z 190,A -164.3385,B 1.0274,C 0.0979,E1 0.8749,E2 257.9144} C_DIS
LIN {X -133.0789,Y -26.8962,Z 190,A -162.4838,B 1.027,C 0.1021,E1 0.8759,E2 256.0041} C_DIS
LIN {X -132.2303,Y -30.8032,Z 190,A -160.5087,B 1.0265,C 0.1068,E1 0.8771,E2 253.992} C_DIS
LIN {X -131.3348,Y -34.4216,Z 190,A -158.5895,B 1.026,C 0.1112,E1 0.8785,E2 252.0277} C_DIS
LIN {X -130.1824,Y -38.5493,Z 190,A -156.5236,B 1.0255,C 0.1161,E1 0.8801,E2 249.9284} C_DIS
LIN {X -129.0507,Y -42.1875,Z 190,A -154.8035,B 1.025,C 0.1204,E1 0.8816,E2 248.194} C_DIS
LIN {X -127.4108,Y -46.9073,Z 190,A -152.1115,B 1.0243,C 0.1261,E1 0.8842,E2 245.4247} C_DIS
LIN {X -125.4663,Y -51.8818,Z 190,A -149.8062,B 1.0236,C 0.1317,E1 0.8866,E2 243.1133} C_DIS
LIN {X -124.0472,Y -55.1874,Z 190,A -148.1302,B 1.0231,C 0.1355,E1 0.8885,E2 241.4165} C_DIS
LIN {X -122.7134,Y -58.0941,Z 190,A -146.5156,B 1.0226,C 0.1389,E1 0.8905,E2 239.7665} C_DIS
LIN {X -121.0228,Y -61.5368,Z 190,A -144.73,B 1.0221,C 0.1428,E1 0.8927,E2 237.9587} C_DIS
LIN {X -118.6402,Y -66.0183,Z 190,A -142.1633,B 1.0214,C 0.1479,E1 0.8962,E2 235.3349} C_DIS
LIN {X -116.4695,Y -69.7766,Z 190,A -140.1861,B 1.0208,C 0.152,E1 0.8991,E2 233.3382} C_DIS
LIN {X -114.196,Y -73.4384,Z 190,A -138.1171,B 1.0202,C 0.156,E1 0.9022,E2 231.2353} C_DIS
LIN {X -111.8392,Y -76.9796,Z 190,A -136.0862,B 1.0196,C 0.1598,E1 0.9055,E2 229.1723} C_DIS
LIN {X -109.281,Y -80.5702,Z 190,A -134.1128,B 1.019,C 0.1637,E1 0.9088,E2 227.1836} C_DIS
LIN {X -106.9595,Y -83.6276,Z 190,A -132.1871,B 1.0185,C 0.1669,E1 0.9121,E2 225.2159} C_DIS
LIN {X -104.1403,Y -87.1129,Z 190,A -130.1246,B 1.0179,C 0.1705,E1 0.9159,E2 223.1299} C_DIS
LIN {X -101.3055,Y -90.394,Z 190,A -128.1981,B 1.0173,C 0.1739,E1 0.9195,E2 221.1901} C_DIS
LIN {X -98.5152,Y -93.4275,Z 190,A -126.1929,B 1.0168,C 0.1769,E1 0.9234,E2 219.148} C_DIS
LIN {X -96.1697,Y -95.8397,Z 190,A -124.2051,B 1.0164,C 0.179,E1 0.9275,E2 217.0805} C_DIS
LIN {X -93.1196,Y -98.8051,Z 190,A -122.5324,B 1.0159,C 0.182,E1 0.9309,E2 215.4251} C_DIS
LIN {X -89.1469,Y -102.4045,Z 190,A -120.2245,B 1.0152,C 0.1855,E1 0.9357,E2 213.1109} C_DIS
LIN {X -85.6312,Y -105.3625,Z 190,A -118.114,B 1.0147,C 0.1882,E1 0.9404,E2 210.9762} C_DIS
LIN {X -82.1118,Y -108.1279,Z 190,A -116.0562,B 1.0143,C 0.1907,E1 0.945,E2 208.8945} C_DIS
LIN {X -77.9276,Y -111.1813,Z 190,A -113.429,B 1.0138,C 0.193,E1 0.9512,E2 206.2045} C_DIS
LIN {X -74.7479,Y -113.3428,Z 190,A -112.091,B 1.0134,C 0.1953,E1 0.9542,E2 204.9067} C_DIS
LIN {X -71.1821,Y -115.6157,Z 190,A -109.8117,B 1.0131,C 0.1966,E1 0.9599,E2 202.5568} C_DIS
LIN {X -67.825,Y -117.6166,Z 190,A -108.4338,B 1.0127,C 0.1987,E1 0.9631,E2 201.2174} C_DIS
LIN {X -63.9366,Y -119.7751,Z 190,A -106.5245,B 1.0124,C 0.2004,E1 0.9679,E2 199.303} C_DIS
LIN {X -60.5966,Y -121.4977,Z 190,A -104.788,B 1.0122,C 0.2016,E1 0.9723,E2 197.5447} C_DIS
LIN {X -54.9417,Y -124.1571,Z 190,A -102.0155,B 1.0118,C 0.2034,E1 0.9795,E2 194.7524} C_DIS
LIN {X -51.6489,Y -125.5636,Z 190,A -100.0477,B 1.0118,C 0.2036,E1 0.9848,E2 192.7187} C_DIS
LIN {X -47.6376,Y -127.1376,Z 190,A -98.643,B 1.0114,C 0.2054,E1 0.9883,E2 191.3729} C_DIS
LIN {X -43.598,Y -128.581,Z 190,A -96.7229,B 1.0113,C 0.2061,E1 0.9935,E2 189.4366} C_DIS
LIN {X -40.0273,Y -129.7353,Z 190,A -95.1421,B 1.0111,C 0.2067,E1 0.9978,E2 187.8556} C_DIS
LIN {X -36.4708,Y -130.7793,Z 190,A -93.7447,B 1.0109,C 0.2076,E1 1.0015,E2 186.4815} C_DIS
LIN {X -33.4807,Y -131.5766,Z 190,A -92.2775,B 1.0109,C 0.2076,E1 1.0056,E2 184.9908} C_DIS
LIN {X -29.7969,Y -132.4602,Z 190,A -90.5876,B 1.0109,C 0.2076,E1 1.0103,E2 183.2872} C_DIS
LIN {X -24.967,Y -133.4553,Z 190,A -88.2924,B 1.0109,C 0.2074,E1 1.0167,E2 180.9604} C_DIS
LIN {X -21.5477,Y -134.0511,Z 190,A -87.0038,B 1.0109,C 0.2078,E1 1.0202,E2 179.6965} C_DIS
LIN {X -17.4311,Y -134.6462,Z 190,A -85.3731,B 1.0109,C 0.208,E1 1.0248,E2 178.0829} C_DIS
LIN {X -14.0421,Y -135.0424,Z 190,A -83.8895,B 1.0109,C 0.2077,E1 1.029,E2 176.5924} C_DIS
LIN {X -6.1621,Y -135.6314,Z 190,A -80.711,B 1.0109,C 0.2073,E1 1.0379,E2 173.4348} C_DIS
LIN {X -0.0585,Y -135.7716,Z 190,A -78.1667,B 1.0112,C 0.2064,E1 1.045,E2 170.8939} C_DIS
LIN {X -0.0585,Y -135.7716,Z 190,A -78.1669,B 1.0112,C 0.2064,E1 1.045,E2 170.8941} C_DIS
Enddeposition()
LIN {X 0.9781,Y -136.665,Z 190,A -78.7414,B 1.1026,C 0.2139,E1 1.1352,E2 171.6119} C_DIS
Startdeposition()
$VEL.CP = VEL_PRINT
LIN {X -5.3713,Y -136.5631,Z 190,A -81.2316,B 1.1026,C 0.2143,E1 1.1282,E2 174.079} C_DIS
LIN {X -9.9278,Y -136.3076,Z 190,A -83.7238,B 1.1021,C 0.2165,E1 1.1209,E2 176.6546} C_DIS
LIN {X -13.1218,Y -136.0372,Z 190,A -84.5683,B 1.1024,C 0.2153,E1 1.1188,E2 177.4287} C_DIS
LIN {X -15.8303,Y -135.7491,Z 190,A -86.1494,B 1.1021,C 0.2166,E1 1.1142,E2 179.0729} C_DIS
LIN {X -20.4874,Y -135.1249,Z 190,A -88.0739,B 1.1021,C 0.2165,E1 1.1088,E2 180.9919} C_DIS
LIN {X -25.9848,Y -134.1759,Z 190,A -90.1963,B 1.1023,C 0.2157,E1 1.103,E2 183.0845} C_DIS
LIN {X -29.007,Y -133.5548,Z 190,A -91.5309,B 1.1023,C 0.2156,E1 1.0993,E2 184.4254} C_DIS
LIN {X -32.212,Y -132.8182,Z 190,A -92.9187,B 1.1023,C 0.2153,E1 1.0955,E2 185.815} C_DIS
LIN {X -35.6342,Y -131.9417,Z 190,A -94.3805,B 1.1024,C 0.2148,E1 1.0915,E2 187.2746} C_DIS
LIN {X -38.5215,Y -131.1272,Z 190,A -95.716,B 1.1025,C 0.2145,E1 1.0878,E2 188.6215} C_DIS
LIN {X -41.9623,Y -130.0674,Z 190,A -97.2579,B 1.1026,C 0.2139,E1 1.0837,E2 190.1686} C_DIS
LIN {X -45.2505,Y -128.9607,Z 190,A -98.7656,B 1.1027,C 0.2132,E1 1.0796,E2 191.6842} C_DIS
LIN {X -48.5385,Y -127.76,Z 190,A -101.1314,B 1.1026,C 0.2142,E1 1.0731,E2 194.1773} C_DIS
LIN {X -54.3182,Y -125.4102,Z 190,A -102.6092,B 1.1033,C 0.2102,E1 1.0696,E2 195.4951} C_DIS
LIN {X -59.2173,Y -123.173,Z 190,A -105.3449,B 1.1035,C 0.2092,E1 1.0625,E2 198.2991} C_DIS
LIN {X -62.8385,Y -121.3676,Z 190,A -107.1317,B 1.1038,C 0.2078,E1 1.0579,E2 200.0991} C_DIS
LIN {X -66.4262,Y -119.4418,Z 190,A -108.9527,B 1.1041,C 0.2063,E1 1.0534,E2 201.9365} C_DIS
LIN {X -73.946,Y -114.9383,Z 190,A -113.4566,B 1.1046,C 0.2033,E1 1.0423,E2 206.5569} C_DIS
LIN {X -78.4345,Y -111.9237,Z 190,A -115.1367,B 1.1053,C 0.1997,E1 1.0386,E2 208.1552} C_DIS
LIN {X -81.606,Y -109.6321,Z 190,A -116.9619,B 1.1056,C 0.1977,E1 1.0344,E2 210.0065} C_DIS
LIN {X -85.1216,Y -106.9254,Z 190,A -118.9663,B 1.1061,C 0.1952,E1 1.0299,E2 212.0312} C_DIS
LIN {X -88.6432,Y -104.0246,Z 190,A -121.039,B 1.1066,C 0.1925,E1 1.0254,E2 214.1262} C_DIS
LIN {X -91.9909,Y -101.0764,Z 190,A -123.5541,B 1.107,C 0.19,E1 1.02,E2 216.7306} C_DIS
LIN {X -95.4388,Y -97.8279,Z 190,A -125.2391,B 1.1076,C 0.1864,E1 1.0167,E2 218.3739} C_DIS
LIN {X -98.706,Y -94.5298,Z 190,A -127.3288,B 1.1081,C 0.1831,E1 1.0125,E2 220.4833} C_DIS
LIN {X -101.6949,Y -91.3067,Z 190,A -129.2936,B 1.1087,C 0.1798,E1 1.0088,E2 222.4648} C_DIS
LIN {X -104.4369,Y -88.1579,Z 190,A -131.2592,B 1.1092,C 0.1765,E1 1.0051,E2 224.4598} C_DIS
LIN {X -107.2489,Y -84.7144,Z 190,A -133.2933,B 1.1098,C 0.1729,E1 1.0015,E2 226.5171} C_DIS
LIN {X -109.9058,Y -81.2379,Z 190,A -135.3313,B 1.1103,C 0.1692,E1 0.998,E2 228.5826} C_DIS
LIN {X -112.4596,Y -77.6641,Z 190,A -137.3564,B 1.1109,C 0.1654,E1 0.9947,E2 230.6324} C_DIS
LIN {X -114.8266,Y -74.1196,Z 190,A -139.3667,B 1.1115,C 0.1615,E1 0.9916,E2 232.6728} C_DIS
LIN {X -117.2477,Y -70.2268,Z 190,A -141.5074,B 1.1121,C 0.1572,E1 0.9884,E2 234.8427} C_DIS
LIN {X -119.9868,Y -65.4358,Z 190,A -144.2167,B 1.1129,C 0.1519,E1 0.9846,E2 237.6047} C_DIS
LIN {X -121.8466,Y -61.8998,Z 190,A -145.8924,B 1.1134,C 0.1479,E1 0.9825,E2 239.28} C_DIS
LIN {X -123.4998,Y -58.5334,Z 190,A -147.6563,B 1.1139,C 0.1441,E1 0.9803,E2 241.0692} C_DIS
LIN {X -124.9427,Y -55.387,Z 190,A -149.278,B 1.1143,C 0.1405,E1 0.9784,E2 242.7133} C_DIS
LIN {X -126.2886,Y -52.2454,Z 190,A -151.0264,B 1.1148,C 0.1369,E1 0.9765,E2 244.5033} C_DIS
LIN {X -128.9428,Y -45.302,Z 190,A -154.2877,B 1.1157,C 0.1289,E1 0.9732,E2 247.7827} C_DIS
LIN {X -129.9499,Y -42.3297,Z 190,A -155.8629,B 1.1161,C 0.1254,E1 0.9718,E2 249.3918} C_DIS
LIN {X -130.8027,Y -39.6109,Z 190,A -157.2367,B 1.1165,C 0.1222,E1 0.9707,E2 250.7888} C_DIS
LIN {X -131.8073,Y -36.1323,Z 190,A -159.1551,B 1.117,C 0.118,E1 0.9692,E2 252.7592} C_DIS
LIN {X -132.8297,Y -32.1641,Z 190,A -160.9385,B 1.1174,C 0.1134,E1 0.968,E2 254.5504} C_DIS
LIN {X -133.6688,Y -28.4786,Z 190,A -162.7271,B 1.1179,C 0.109,E1 0.9669,E2 256.3649} C_DIS
LIN {X -134.3075,Y -25.2961,Z 190,A -164.2673,B 1.1182,C 0.1052,E1 0.966,E2 257.9278} C_DIS
LIN {X -134.8282,Y -22.3526,Z 190,A -165.7423,B 1.1186,C 0.1017,E1 0.9653,E2 259.4309} C_DIS
LIN {X -135.3164,Y -19.1778,Z 190,A -167.3299,B 1.1189,C 0.0978,E1 0.9647,E2 261.049} C_DIS
LIN {X -135.8685,Y -14.7674,Z 190,A -169.5247,B 1.1194,C 0.0925,E1 0.9639,E2 263.2856} C_DIS
LIN {X -136.2817,Y -10.2823,Z 190,A -171.6462,B 1.1198,C 0.0871,E1 0.9634,E2 265.4359} C_DIS
LIN {X -136.517,Y -6.4502,Z 190,A -173.441,B 1.1201,C 0.0825,E1 0.9631,E2 267.2535} C_DIS
LIN {X -136.6416,Y -2.7643,Z 190,A -175.2926,B 1.1205,C 0.078,E1 0.963,E2 269.143} C_DIS
LIN {X -136.6653,Y 1.0004,Z 190,A -177.1403,B 1.1208,C 0.0734,E1 0.963,E2 271.0238} C_DIS
LIN {X -136.5631,Y 5.371,Z 190,A -179.1872,B 1.1211,C 0.0681,E1 0.9632,E2 273.0966} C_DIS
LIN {X -136.3151,Y 9.825,Z 190,A 178.6649,B 1.1214,C 0.0627,E1 0.9636,E2 275.2782} C_DIS
LIN {X -135.9663,Y 13.8587,Z 190,A 176.5741,B 1.1217,C 0.0577,E1 0.9641,E2 277.417} C_DIS
LIN {X -135.4582,Y 18.1523,Z 190,A 174.6896,B 1.1219,C 0.0527,E1 0.9648,E2 279.3093} C_DIS
LIN {X -134.87,Y 22.1024,Z 190,A 172.7003,B 1.1221,C 0.0478,E1 0.9657,E2 281.3364} C_DIS
LIN {X -134.2363,Y 25.6686,Z 190,A 170.9666,B 1.1223,C 0.0435,E1 0.9666,E2 283.0956} C_DIS
LIN {X -133.0394,Y 31.2941,Z 190,A 168.3277,B 1.1226,C 0.0368,E1 0.9682,E2 285.7609} C_DIS
LIN {X -131.8324,Y 36.0428,Z 190,A 165.9648,B 1.1227,C 0.0311,E1 0.9698,E2 288.1601} C_DIS
LIN {X -131.0242,Y 38.873,Z 190,A 164.4972,B 1.1228,C 0.0277,E1 0.971,E2 289.6551} C_DIS
LIN {X -130.1023,Y 41.853,Z 190,A 163.0274,B 1.1229,C 0.0242,E1 0.9723,E2 291.1437} C_DIS
LIN {X -129.0128,Y 45.1003,Z 190,A 161.4203,B 1.1229,C 0.0204,E1 0.9737,E2 292.7704} C_DIS
LIN {X -127.7717,Y 48.5073,Z 190,A 159.6928,B 1.123,C 0.0163,E1 0.9754,E2 294.5218} C_DIS
LIN {X -126.5151,Y 51.6966,Z 190,A 157.8965,B 1.123,C 0.0125,E1 0.9774,E2 296.3599} C_DIS
LIN {X -125.0676,Y 55.1076,Z 190,A 156.1611,B 1.1231,C 0.0086,E1 0.9793,E2 298.1159} C_DIS
LIN {X -123.5517,Y 58.4246,Z 190,A 154.4382,B 1.1231,C 0.0047,E1 0.9814,E2 299.8606} C_DIS
LIN {X -121.4383,Y 62.7018,Z 190,A 151.8846,B 1.1231,C -0.0003,E1 0.9847,E2 302.4777} C_DIS
LIN {X -119.6614,Y 66.0296,Z 190,A 150.7429,B 1.1231,C -0.0039,E1 0.9862,E2 303.567} C_DIS
LIN {X -118.0577,Y 68.856,Z 190,A 148.8335,B 1.1231,C -0.0072,E1 0.9889,E2 305.5393} C_DIS
LIN {X -115.65,Y 72.8273,Z 190,A 146.7653,B 1.1231,C -0.0116,E1 0.992,E2 307.6204} C_DIS
LIN {X -113.4495,Y 76.2108,Z 190,A 144.827,B 1.1231,C -0.0154,E1 0.995,E2 309.586} C_DIS
LIN {X -110.9083,Y 79.8639,Z 190,A 142.7955,B 1.1231,C -0.0194,E1 0.9983,E2 311.6354} C_DIS
LIN {X -108.7536,Y 82.7737,Z 190,A 141.2506,B 1.1229,C -0.0226,E1 1.0009,E2 313.1824} C_DIS
LIN {X -106.4077,Y 85.7679,Z 190,A 138.695,B 1.1229,C -0.0258,E1 1.0056,E2 315.846} C_DIS
LIN {X -102.9752,Y 89.8601,Z 190,A 136.6983,B 1.1228,C -0.0301,E1 1.0092,E2 317.814} C_DIS
LIN {X -98.4305,Y 94.8171,Z 190,A 133.9978,B 1.1226,C -0.0354,E1 1.0144,E2 320.4993} C_DIS
LIN {X -92.8455,Y 100.2924,Z 190,A 130.4936,B 1.1224,C -0.0409,E1 1.0215,E2 324.027} C_DIS
LIN {X -88.8016,Y 103.89,Z 190,A 127.9782,B 1.1223,C -0.0445,E1 1.0269,E2 326.5688} C_DIS
LIN {X -86.1149,Y 106.1278,Z 190,A 125.7664,B 1.1223,C -0.0463,E1 1.0319,E2 328.8625} C_DIS
LIN {X -82.6992,Y 108.8091,Z 190,A 124.074,B 1.1221,C -0.049,E1 1.0356,E2 330.5397} C_DIS
LIN {X -78.1062,Y 112.1523,Z 190,A 121.7296,B 1.122,C -0.0523,E1 1.041,E2 332.8786} C_DIS
LIN {X -74.3958,Y 114.6473,Z 190,A 119.3809,B 1.1219,C -0.0542,E1 1.0466,E2 335.2783} C_DIS
LIN {X -71.008,Y 116.7763,Z 190,A 118.2271,B 1.1217,C -0.0566,E1 1.0492,E2 336.3735} C_DIS
LIN {X -68.3026,Y 118.3788,Z 190,A 116.2876,B 1.1217,C -0.0575,E1 1.0541,E2 338.3806} C_DIS
LIN {X -65.0913,Y 120.1749,Z 190,A 114.9185,B 1.1217,C -0.0592,E1 1.0575,E2 339.7299} C_DIS
LIN {X -61.2945,Y 122.1548,Z 190,A 113.1749,B 1.1215,C -0.061,E1 1.0618,E2 341.4667} C_DIS
LIN {X -57.9537,Y 123.7739,Z 190,A 111.1368,B 1.1215,C -0.0617,E1 1.0671,E2 343.5566} C_DIS
LIN {X -54.5367,Y 125.3157,Z 190,A 109.7381,B 1.1214,C -0.0632,E1 1.0707,E2 344.9355} C_DIS
LIN {X -49.8813,Y 127.2407,Z 190,A 107.3866,B 1.1214,C -0.0643,E1 1.0769,E2 347.312} C_DIS
LIN {X -46.6019,Y 128.4777,Z 190,A 105.7457,B 1.1213,C -0.0649,E1 1.0813,E2 348.9707} C_DIS
LIN {X -42.5547,Y 129.8759,Z 190,A 104.4027,B 1.1212,C -0.0665,E1 1.0848,E2 350.2637} C_DIS
LIN {X -39.7219,Y 130.7688,Z 190,A 103.1695,B 1.1212,C -0.0671,E1 1.0881,E2 351.495} C_DIS
LIN {X -36.1855,Y 131.7925,Z 190,A 101.3829,B 1.1212,C -0.0673,E1 1.093,E2 353.3073} C_DIS
LIN {X -32.2049,Y 132.8199,Z 190,A 99.7535,B 1.1212,C -0.068,E1 1.0974,E2 354.9256} C_DIS
LIN {X -28.7911,Y 133.6014,Z 190,A 98.3308,B 1.1211,C -0.0684,E1 1.1013,E2 356.3426} C_DIS
LIN {X -25.3584,Y 134.2956,Z 190,A 96.8123,B 1.1211,C -0.0684,E1 1.1056,E2 357.8659} C_DIS
LIN {X -18.0162,Y 135.4761,Z 190,A 93.6391,B 1.1211,C -0.0684,E1 1.1144,E2 361.0438} C_DIS
LIN {X -13.4747,Y 136.0033,Z 190,A 91.8776,B 1.1211,C -0.0687,E1 1.1193,E2 362.7875} C_DIS
LIN {X -4.6702,Y 136.5904,Z 190,A 87.1339,B 1.1213,C -0.0652,E1 1.133,E2 367.6425} C_DIS
LIN {X 2.3991,Y 136.6477,Z 190,A 85.5184,B 1.1211,C -0.0675,E1 1.1371,E2 369.1109} C_DIS
LIN {X 9.5227,Y 136.3371,Z 190,A 82.4662,B 1.1212,C -0.0658,E1 1.1458,E2 372.1692} C_DIS
LIN {X 14.6089,Y 135.8855,Z 190,A 80.2206,B 1.1213,C -0.0641,E1 1.1521,E2 374.4256} C_DIS
LIN {X 18.2068,Y 135.4511,Z 190,A 78.6321,B 1.1214,C -0.0628,E1 1.1565,E2 376.0212} C_DIS
LIN {X 22.5462,Y 134.7959,Z 190,A 76.9984,B 1.1214,C -0.062,E1 1.161,E2 377.6318} C_DIS
LIN {X 25.7831,Y 134.2144,Z 190,A 75.6749,B 1.1215,C -0.0609,E1 1.1647,E2 378.9489} C_DIS
LIN {X 28.991,Y 133.5582,Z 190,A 74.3586,B 1.1215,C -0.0598,E1 1.1683,E2 380.2585} C_DIS
LIN {X 32.5181,Y 132.7444,Z 190,A 72.8565,B 1.1217,C -0.0584,E1 1.1724,E2 381.7586} C_DIS
LIN {X 36.7079,Y 131.6464,Z 190,A 71.165,B 1.1217,C -0.0568,E1 1.177,E2 383.4358} C_DIS
LIN {X 40.3518,Y 130.576,Z 190,A 69.641,B 1.1218,C -0.0552,E1 1.181,E2 384.952} C_DIS
LIN {X 43.944,Y 129.4132,Z 190,A 68.156,B 1.1218,C -0.0536,E1 1.185,E2 386.4258} C_DIS
LIN {X 51.0882,Y 126.7603,Z 190,A 65.1911,B 1.122,C -0.0503,E1 1.1927,E2 389.3645} C_DIS
LIN {X 56.1133,Y 124.6178,Z 190,A 62.9932,B 1.1222,C -0.0474,E1 1.1984,E2 391.5517} C_DIS
LIN {X 59.2598,Y 123.1527,Z 190,A 61.628,B 1.1222,C -0.0456,E1 1.2018,E2 392.9067} C_DIS
LIN {X 62.1039,Y 121.7427,Z 190,A 60.3722,B 1.1223,C -0.0438,E1 1.205,E2 394.1539} C_DIS
LIN {X 65.4164,Y 119.9976,Z 190,A 58.2118,B 1.1225,C -0.0389,E1 1.2105,E2 396.3802} C_DIS
LIN {X 70.4316,Y 117.1249,Z 190,A 56.5607,B 1.1225,C -0.0379,E1 1.2142,E2 397.9448} C_DIS
LIN {X 75.1322,Y 114.166,Z 190,A 54.4242,B 1.1226,C -0.0346,E1 1.2192,E2 400.0593} C_DIS
LIN {X 78.8104,Y 111.6586,Z 190,A 52.709,B 1.1227,C -0.0318,E1 1.2232,E2 401.7573} C_DIS
LIN {X 82.5321,Y 108.9369,Z 190,A 50.9102,B 1.1228,C -0.0287,E1 1.2272,E2 403.5407} C_DIS
LIN {X 86.0782,Y 106.1574,Z 190,A 49.1793,B 1.1228,C -0.0257,E1 1.2309,E2 405.2537} C_DIS
LIN {X 89.5404,Y 103.2541,Z 190,A 47.4805,B 1.1229,C -0.0228,E1 1.2345,E2 406.93} C_DIS
LIN {X 92.5249,Y 100.5876,Z 190,A 45.9271,B 1.1229,C -0.0199,E1 1.2377,E2 408.4691} C_DIS
LIN {X 95.5341,Y 97.7344,Z 190,A 44.3117,B 1.123,C -0.0168,E1 1.241,E2 410.0704} C_DIS
LIN {X 98.7864,Y 94.4456,Z 190,A 42.5659,B 1.123,C -0.0134,E1 1.2443,E2 411.7939} C_DIS
LIN {X 101.877,Y 91.1033,Z 190,A 40.8378,B 1.1231,C -0.01,E1 1.2475,E2 413.5013} C_DIS
LIN {X 104.9111,Y 87.5927,Z 190,A 39.0573,B 1.1231,C -0.0064,E1 1.2507,E2 415.2628} C_DIS
LIN {X 107.6678,Y 84.1811,Z 190,A 37.4482,B 1.1231,C -0.0033,E1 1.2535,E2 416.8451} C_DIS
LIN {X 110.2308,Y 80.7955,Z 190,A 35.783,B 1.1231,C 0.0004,E1 1.2563,E2 418.4971} C_DIS
LIN {X 112.9147,Y 77.001,Z 190,A 33.616,B 1.1231,C 0.0062,E1 1.2598,E2 420.6903} C_DIS
LIN {X 115.4973,Y 73.0694,Z 190,A 32.2574,B 1.1231,C 0.008,E1 1.2617,E2 421.9767} C_DIS
LIN {X 118.5984,Y 67.9205,Z 190,A 30.1337,B 1.1231,C 0.0122,E1 1.2647,E2 424.0537} C_DIS
LIN {X 120.3285,Y 64.8058,Z 190,A 28.7007,B 1.1231,C 0.0157,E1 1.2666,E2 425.4798} C_DIS
LIN {X 121.9259,Y 61.744,Z 190,A 27.453,B 1.1231,C 0.0183,E1 1.2681,E2 426.7037} C_DIS
LIN {X 123.341,Y 58.8657,Z 190,A 25.5741,B 1.1229,C 0.0246,E1 1.2705,E2 428.6472} C_DIS
LIN {X 125.7284,Y 53.5823,Z 190,A 24.0666,B 1.1229,C 0.0261,E1 1.272,E2 430.0443} C_DIS
LIN {X 128.4444,Y 46.6944,Z 190,A 21.2549,B 1.1227,C 0.0328,E1 1.2749,E2 432.8215} C_DIS
LIN {X 129.7185,Y 43.0273,Z 190,A 19.8543,B 1.1226,C 0.036,E1 1.2761,E2 434.1948} C_DIS
LIN {X 130.7456,Y 39.7974,Z 190,A 18.5399,B 1.1225,C 0.0392,E1 1.2772,E2 435.4967} C_DIS
LIN {X 131.6198,Y 36.8031,Z 190,A 17.4077,B 1.1224,C 0.0418,E1 1.278,E2 436.6077} C_DIS
LIN {X 132.5597,Y 33.2612,Z 190,A 16.0564,B 1.1223,C 0.045,E1 1.2789,E2 437.9367} C_DIS
LIN {X 133.268,Y 30.297,Z 190,A 14.879,B 1.1221,C 0.0479,E1 1.2797,E2 439.1023} C_DIS
LIN {X 134.0652,Y 26.5571,Z 190,A 13.4802,B 1.122,C 0.0512,E1 1.2805,E2 440.4763} C_DIS
LIN {X 134.7612,Y 22.7546,Z 190,A 11.9398,B 1.1218,C 0.0553,E1 1.2812,E2 442.0074} C_DIS
LIN {X 135.4279,Y 18.3838,Z 190,A 9.7158,B 1.1214,C 0.0625,E1 1.2821,E2 444.2785} C_DIS
LIN {X 136.0755,Y 12.7227,Z 190,A 8.009,B 1.1213,C 0.0654,E1 1.2825,E2 445.9013} C_DIS
LIN {X 136.3374,Y 9.5185,Z 190,A 6.7122,B 1.1211,C 0.0688,E1 1.2828,E2 447.1924} C_DIS
LIN {X 136.5489,Y 5.7339,Z 190,A 5.7847,B 1.1211,C 0.0696,E1 1.2828,E2 448.037} C_DIS
LIN {X 136.668,Y 0.4423,Z 190,A 3.4871,B 1.1206,C 0.0762,E1 1.283,E2 450.3459} C_DIS
LIN {X 136.4522,Y -7.7182,Z 190,A 0.5331,B 1.1201,C 0.0831,E1 1.2827,E2 453.2421} C_DIS
LIN {X 136.2435,Y -10.7943,Z 190,A -1.3797,B 1.1195,C 0.0903,E1 1.2823,E2 455.2349} C_DIS
LIN {X 135.5247,Y -17.6451,Z 190,A -3.1228,B 1.1195,C 0.0918,E1 1.2817,E2 456.8329} C_DIS
LIN {X 134.9642,Y -21.5248,Z 190,A -4.6636,B 1.1191,C 0.0958,E1 1.281,E2 458.3615} C_DIS
LIN {X 134.2292,Y -25.7055,Z 190,A -6.1319,B 1.1188,C 0.099,E1 1.2803,E2 459.7904} C_DIS
LIN {X 133.5591,Y -28.987,Z 190,A -7.4201,B 1.1185,C 0.1022,E1 1.2796,E2 461.0643} C_DIS
LIN {X 132.8192,Y -32.2077,Z 190,A -8.6121,B 1.1183,C 0.1049,E1 1.2788,E2 462.232} C_DIS
LIN {X 132.0107,Y -35.3757,Z 190,A -9.8164,B 1.118,C 0.1077,E1 1.278,E2 463.4153} C_DIS
LIN {X 131.0508,Y -38.7823,Z 190,A -11.135,B 1.1177,C 0.1108,E1 1.277,E2 464.7132} C_DIS
LIN {X 128.3588,Y -46.9318,Z 190,A -14.372,B 1.1169,C 0.1184,E1 1.2742,E2 467.9051} C_DIS
LIN {X 127.0855,Y -50.2806,Z 190,A -16.2533,B 1.1162,C 0.1245,E1 1.2722,E2 469.8376} C_DIS
LIN {X 125.2229,Y -54.7515,Z 190,A -17.5323,B 1.1162,C 0.1257,E1 1.2709,E2 471.0183} C_DIS
LIN {X 123.7413,Y -58.0242,Z 190,A -18.8888,B 1.1158,C 0.1287,E1 1.2693,E2 472.3561} C_DIS
LIN {X 122.4043,Y -60.7905,Z 190,A -20.0722,B 1.1154,C 0.1315,E1 1.2679,E2 473.5263} C_DIS
LIN {X 120.9232,Y -63.685,Z 190,A -21.2621,B 1.1151,C 0.134,E1 1.2664,E2 474.6939} C_DIS
LIN {X 118.9009,Y -67.3903,Z 190,A -22.9412,B 1.1147,C 0.138,E1 1.2641,E2 476.3623} C_DIS
LIN {X 115.8313,Y -72.5396,Z 190,A -25.1811,B 1.1141,C 0.1427,E1 1.2609,E2 478.5672} C_DIS
LIN {X 112.7541,Y -77.2347,Z 190,A -27.414,B 1.1134,C 0.1478,E1 1.2575,E2 480.7855} C_DIS
LIN {X 110.2676,Y -80.7454,Z 190,A -29.4386,B 1.1127,C 0.1532,E1 1.2541,E2 482.8414} C_DIS
LIN {X 107.1737,Y -84.8097,Z 190,A -30.8559,B 1.1125,C 0.1544,E1 1.2518,E2 484.1621} C_DIS
LIN {X 104.4743,Y -88.1133,Z 190,A -32.4727,B 1.1121,C 0.1576,E1 1.2489,E2 485.7568} C_DIS
LIN {X 101.109,Y -91.955,Z 190,A -34.2823,B 1.1116,C 0.1607,E1 1.2457,E2 487.5226} C_DIS
LIN {X 98.1619,Y -95.0945,Z 190,A -36.0379,B 1.1111,C 0.1644,E1 1.2423,E2 489.2728} C_DIS
LIN {X 95.3337,Y -97.9303,Z 190,A -37.6738,B 1.1106,C 0.1678,E1 1.239,E2 490.904} C_DIS
LIN {X 92.1517,Y -100.9305,Z 190,A -39.4605,B 1.11,C 0.1713,E1 1.2354,E2 492.6857} C_DIS
LIN {X 87.3696,Y -105.0969,Z 190,A -41.6274,B 1.1096,C 0.1743,E1 1.2309,E2 494.7866} C_DIS
LIN {X 84.5512,Y -107.3772,Z 190,A -43.1736,B 1.1091,C 0.1774,E1 1.2275,E2 496.3376} C_DIS
LIN {X 81.0736,Y -110.0265,Z 190,A -44.9752,B 1.1085,C 0.1807,E1 1.2234,E2 498.1363} C_DIS
LIN {X 75.6975,Y -113.7922,Z 190,A -47.1411,B 1.1082,C 0.183,E1 1.2186,E2 500.2227} C_DIS
LIN {X 71.1422,Y -116.6943,Z 190,A -49.8677,B 1.1071,C 0.189,E1 1.212,E2 503.0155} C_DIS
LIN {X 67.3296,Y -118.9349,Z 190,A -51.1102,B 1.1071,C 0.1893,E1 1.2092,E2 504.174} C_DIS
LIN {X 65.1532,Y -120.1412,Z 190,A -52.2062,B 1.1068,C 0.1912,E1 1.2064,E2 505.2782} C_DIS
LIN {X 61.8114,Y -121.8916,Z 190,A -53.5932,B 1.1065,C 0.1928,E1 1.203,E2 506.639} C_DIS
LIN {X 58.0629,Y -123.7233,Z 190,A -55.2786,B 1.1061,C 0.1952,E1 1.1988,E2 508.3168} C_DIS
LIN {X 52.4806,Y -126.1904,Z 190,A -57.9205,B 1.1054,C 0.1992,E1 1.1919,E2 510.9721} C_DIS
LIN {X 49.3017,Y -127.466,Z 190,A -58.9173,B 1.1054,C 0.1992,E1 1.1895,E2 511.9082} C_DIS
LIN {X 46.4846,Y -128.52,Z 190,A -60.1546,B 1.1051,C 0.2008,E1 1.1862,E2 513.143} C_DIS
LIN {X 42.2221,Y -129.9844,Z 190,A -61.8975,B 1.1048,C 0.2025,E1 1.1816,E2 514.8666} C_DIS
LIN {X 37.7858,Y -131.3426,Z 190,A -63.7817,B 1.1044,C 0.2045,E1 1.1765,E2 516.7434} C_DIS
LIN {X 34.9179,Y -132.1328,Z 190,A -64.9505,B 1.1042,C 0.2055,E1 1.1734,E2 517.902} C_DIS
LIN {X 32.0052,Y -132.868,Z 190,A -66.2466,B 1.1039,C 0.2069,E1 1.1698,E2 519.204} C_DIS
LIN {X 28.2714,Y -133.7136,Z 190,A -67.7295,B 1.1037,C 0.208,E1 1.1658,E2 520.6707} C_DIS
LIN {X 25.3698,Y -134.2934,Z 190,A -68.9859,B 1.1035,C 0.2092,E1 1.1623,E2 521.9301} C_DIS
LIN {X 16.3905,Y -135.6823,Z 190,A -73.5097,B 1.1025,C 0.2147,E1 1.1494,E2 526.557} C_DIS
LIN {X 9.6526,Y -136.3277,Z 190,A -75.2939,B 1.1028,C 0.2128,E1 1.1448,E2 528.1939} C_DIS
LIN {X 6.5946,Y -136.5097,Z 190,A -77.2135,B 1.1023,C 0.2156,E1 1.1391,E2 530.2044} C_DIS
LIN {X 1.5003,Y -136.6625,Z 190,A -78.7107,B 1.1025,C 0.2145,E1 1.1351,E2 531.6122} C_DIS
LIN {X 1.5003,Y -136.6625,Z 190,A -78.7107,B 1.1025,C 0.2145,E1 1.1351,E2 531.6122} C_DIS
Enddeposition()
LIN {X 0.983,Y -137.5643,Z 190,A -78.8458,B 1.1286,C 0.216,E1 1.1609,E2 531.754} C_DIS
Startdeposition()
$VEL.CP = VEL_PRINT
LIN {X 4.0168,Y -137.5091,Z 190,A -77.1927,B 1.129,C 0.2142,E1 1.1657,E2 530.0442} C_DIS
LIN {X 8.2024,Y -137.323,Z 190,A -75.5308,B 1.129,C 0.2135,E1 1.1704,E2 528.3934} C_DIS
LIN {X 13.5291,Y -136.9011,Z 190,A -73.0628,B 1.1295,C 0.2113,E1 1.1774,E2 525.8891} C_DIS
LIN {X 16.9376,Y -136.5223,Z 190,A -71.3953,B 1.1299,C 0.2093,E1 1.1822,E2 524.1861} C_DIS
LIN {X 21.8763,Y -135.8188,Z 190,A -69.8472,B 1.1299,C 0.2097,E1 1.1863,E2 522.7134} C_DIS
LIN {X 24.8099,Y -135.3129,Z 190,A -68.4698,B 1.1301,C 0.2081,E1 1.1902,E2 521.3153} C_DIS
LIN {X 28.2297,Y -134.6421,Z 190,A -67.2088,B 1.1302,C 0.2075,E1 1.1936,E2 520.0809} C_DIS
LIN {X 32.1374,Y -133.7608,Z 190,A -65.8562,B 1.1302,C 0.2071,E1 1.1972,E2 518.7726} C_DIS
LIN {X 34.7515,Y -133.1074,Z 190,A -64.5876,B 1.1306,C 0.2053,E1 1.2007,E2 517.4824} C_DIS
LIN {X 38.5087,Y -132.0675,Z 190,A -63.1527,B 1.1308,C 0.2043,E1 1.2045,E2 516.0734} C_DIS
LIN {X 41.7756,Y -131.0707,Z 190,A -61.6988,B 1.1311,C 0.2025,E1 1.2084,E2 514.614} C_DIS
LIN {X 45.5285,Y -129.8157,Z 190,A -60.1017,B 1.1314,C 0.2007,E1 1.2126,E2 513.0231} C_DIS
LIN {X 50.1356,Y -128.1063,Z 190,A -57.6685,B 1.1322,C 0.1963,E1 1.2192,E2 510.533} C_DIS
LIN {X 55.161,Y -126.0251,Z 190,A -56.181,B 1.1322,C 0.1965,E1 1.2227,E2 509.1556} C_DIS
LIN {X 58.951,Y -124.2965,Z 190,A -54.6301,B 1.1325,C 0.1948,E1 1.2266,E2 507.6296} C_DIS
LIN {X 62.1351,Y -122.7355,Z 190,A -53.1904,B 1.1328,C 0.1927,E1 1.2302,E2 506.1942} C_DIS
LIN {X 65.4996,Y -120.9761,Z 190,A -51.1833,B 1.1336,C 0.1882,E1 1.2354,E2 504.1252} C_DIS
LIN {X 69.4756,Y -118.7368,Z 190,A -49.7907,B 1.1337,C 0.1875,E1 1.2386,E2 502.8036} C_DIS
LIN {X 73.4384,Y -116.3273,Z 190,A -48.0263,B 1.1341,C 0.1849,E1 1.2427,E2 501.0616} C_DIS
LIN {X 77.9538,Y -113.351,Z 190,A -45.9857,B 1.1346,C 0.1819,E1 1.2474,E2 499.0493} C_DIS
LIN {X 81.2249,Y -111.0307,Z 190,A -44.3998,B 1.135,C 0.1792,E1 1.251,E2 497.4741} C_DIS
LIN {X 84.6038,Y -108.4786,Z 190,A -42.7294,B 1.1355,C 0.1763,E1 1.2547,E2 495.8155} C_DIS
LIN {X 88.0497,Y -105.7008,Z 190,A -41.2765,B 1.1358,C 0.1746,E1 1.2577,E2 494.4161} C_DIS
LIN {X 89.9821,Y -104.0602,Z 190,A -40.1123,B 1.1362,C 0.1719,E1 1.2603,E2 493.236} C_DIS
LIN {X 93.1928,Y -101.1946,Z 190,A -38.4672,B 1.1366,C 0.169,E1 1.2636,E2 491.6102} C_DIS
LIN {X 96.435,Y -98.1099,Z 190,A -36.7802,B 1.1371,C 0.1659,E1 1.267,E2 489.9464} C_DIS
LIN {X 99.2834,Y -95.2265,Z 190,A -35.2058,B 1.1375,C 0.1629,E1 1.27,E2 488.3867} C_DIS
LIN {X 102.1083,Y -92.1914,Z 190,A -33.6351,B 1.1379,C 0.1599,E1 1.273,E2 486.8364} C_DIS
LIN {X 104.8327,Y -89.0805,Z 190,A -32.086,B 1.1383,C 0.1569,E1 1.2758,E2 485.3101} C_DIS
LIN {X 107.5452,Y -85.7863,Z 190,A -30.6355,B 1.1387,C 0.1546,E1 1.2783,E2 483.9036} C_DIS
LIN {X 109.7033,Y -83.0084,Z 190,A -28.7985,B 1.1394,C 0.1491,E1 1.2815,E2 482.0139} C_DIS
LIN {X 112.1711,Y -79.6434,Z 190,A -26.889,B 1.14,C 0.144,E1 1.2846,E2 480.0792} C_DIS
LIN {X 115.6325,Y -74.5288,Z 190,A -25.4312,B 1.14,C 0.144,E1 1.2866,E2 478.7738} C_DIS
LIN {X 118.2903,Y -70.2331,Z 190,A -23.3307,B 1.1407,C 0.1387,E1 1.2897,E2 476.6722} C_DIS
LIN {X 120.3887,Y -66.5718,Z 190,A -21.8137,B 1.1411,C 0.1356,E1 1.2917,E2 475.1869} C_DIS
LIN {X 122.2584,Y -63.0722,Z 190,A -20.2383,B 1.1415,C 0.1318,E1 1.2937,E2 473.6208} C_DIS
LIN {X 123.8493,Y -59.887,Z 190,A -19.0531,B 1.1418,C 0.1297,E1 1.2951,E2 472.4751} C_DIS
LIN {X 125.1404,Y -57.1402,Z 190,A -17.8429,B 1.1421,C 0.1267,E1 1.2966,E2 471.2713} C_DIS
LIN {X 126.922,Y -53.0614,Z 190,A -16.3424,B 1.1424,C 0.1239,E1 1.2982,E2 469.8173} C_DIS
LIN {X 128.1665,Y -49.9808,Z 190,A -15.0117,B 1.1428,C 0.1205,E1 1.2995,E2 468.4927} C_DIS
LIN {X 129.3005,Y -46.9702,Z 190,A -13.9148,B 1.143,C 0.1183,E1 1.3006,E2 467.4277} C_DIS
LIN {X 130.0298,Y -44.9108,Z 190,A -12.6319,B 1.1435,C 0.1138,E1 1.3018,E2 466.0939} C_DIS
LIN {X 131.1566,Y -41.5067,Z 190,A -11.5091,B 1.1436,C 0.1119,E1 1.3027,E2 465.0201} C_DIS
LIN {X 132.3707,Y -37.4554,Z 190,A -9.9729,B 1.144,C 0.1084,E1 1.3039,E2 463.5129} C_DIS
LIN {X 133.2833,Y -34.0643,Z 190,A -8.7821,B 1.1442,C 0.106,E1 1.3047,E2 462.3575} C_DIS
LIN {X 133.9267,Y -31.4492,Z 190,A -7.5688,B 1.1445,C 0.1024,E1 1.3055,E2 461.1313} C_DIS
LIN {X 134.7768,Y -27.5682,Z 190,A -6.2265,B 1.1448,C 0.0996,E1 1.3062,E2 459.8293} C_DIS
LIN {X 135.4557,Y -24.0119,Z 190,A -4.8424,B 1.1451,C 0.0962,E1 1.3069,E2 458.4608} C_DIS
LIN {X 136.4606,Y -17.4212,Z 190,A -2.3965,B 1.1455,C 0.0904,E1 1.3079,E2 456.057} C_DIS
LIN {X 136.8973,Y -13.5686,Z 190,A -0.8479,B 1.1459,C 0.0863,E1 1.3083,E2 454.5161} C_DIS
LIN {X 137.2801,Y -8.8993,Z 190,A 0.641,B 1.1461,C 0.0835,E1 1.3087,E2 453.0867} C_DIS
LIN {X 137.4135,Y -6.5194,Z 190,A 2.0247,B 1.1464,C 0.0784,E1 1.3088,E2 451.6511} C_DIS
LIN {X 137.5439,Y -2.5687,Z 190,A 3.0624,B 1.1464,C 0.0774,E1 1.3089,E2 450.6922} C_DIS
LIN {X 137.5399,Y 2.8106,Z 190,A 5.2337,B 1.1469,C 0.0715,E1 1.3089,E2 448.5287} C_DIS
LIN {X 137.4278,Y 6.2348,Z 190,A 6.8766,B 1.1472,C 0.0663,E1 1.3086,E2 446.857} C_DIS
LIN {X 137.1368,Y 10.8987,Z 190,A 8.2016,B 1.1472,C 0.0644,E1 1.3084,E2 445.6115} C_DIS
LIN {X 136.5737,Y 16.5067,Z 190,A 10.44,B 1.1476,C 0.0585,E1 1.3077,E2 443.3861} C_DIS
LIN {X 136.0606,Y 20.3165,Z 190,A 11.9562,B 1.1478,C 0.0545,E1 1.3071,E2 441.8801} C_DIS
LIN {X 135.4979,Y 23.776,Z 190,A 12.9371,B 1.1478,C 0.0532,E1 1.3067,E2 440.9598} C_DIS
LIN {X 134.8509,Y 27.204,Z 190,A 14.0872,B 1.148,C 0.0509,E1 1.3061,E2 439.8475} C_DIS
LIN {X 134.3467,Y 29.5982,Z 190,A 15.2755,B 1.1481,C 0.0471,E1 1.3053,E2 438.6373} C_DIS
LIN {X 133.4271,Y 33.4973,Z 190,A 16.6369,B 1.1482,C 0.0443,E1 1.3045,E2 437.3141} C_DIS
LIN {X 132.5706,Y 36.7406,Z 190,A 17.8928,B 1.1484,C 0.0412,E1 1.3036,E2 436.0755} C_DIS
LIN {X 131.7369,Y 39.6301,Z 190,A 19.0916,B 1.1484,C 0.0382,E1 1.3026,E2 434.8829} C_DIS
LIN {X 130.5844,Y 43.272,Z 190,A 20.3794,B 1.1485,C 0.0355,E1 1.3015,E2 433.6325} C_DIS
LIN {X 129.5259,Y 46.3451,Z 190,A 21.4858,B 1.1486,C 0.0333,E1 1.3005,E2 432.5565} C_DIS
LIN {X 128.193,Y 49.9126,Z 190,A 23.1176,B 1.1487,C 0.0288,E1 1.2989,E2 430.9184} C_DIS
LIN {X 126.6477,Y 53.718,Z 190,A 24.6491,B 1.1488,C 0.0253,E1 1.2973,E2 429.4088} C_DIS
LIN {X 125.5247,Y 56.2873,Z 190,A 25.8897,B 1.1488,C 0.0218,E1 1.2959,E2 428.1587} C_DIS
LIN {X 123.5489,Y 60.5021,Z 190,A 27.3042,B 1.1489,C 0.0196,E1 1.2942,E2 426.8085} C_DIS
LIN {X 122.033,Y 63.5049,Z 190,A 28.6925,B 1.1489,C 0.0161,E1 1.2925,E2 425.4214} C_DIS
LIN {X 120.0601,Y 67.1632,Z 190,A 30.1191,B 1.149,C 0.0133,E1 1.2906,E2 424.0318} C_DIS
LIN {X 118.3993,Y 70.0502,Z 190,A 31.5921,B 1.149,C 0.0094,E1 1.2885,E2 422.5479} C_DIS
LIN {X 116.0325,Y 73.9039,Z 190,A 33.0851,B 1.149,C 0.0068,E1 1.2864,E2 421.1021} C_DIS
LIN {X 113.9211,Y 77.1182,Z 190,A 34.6965,B 1.149,C 0.0028,E1 1.2839,E2 419.4892} C_DIS
LIN {X 111.2338,Y 80.9466,Z 190,A 36.4491,B 1.149,C -0.0008,E1 1.2811,E2 417.76} C_DIS
LIN {X 108.5922,Y 84.4572,Z 190,A 38.1454,B 1.149,C -0.0045,E1 1.2782,E2 416.0794} C_DIS
LIN {X 105.6619,Y 88.0964,Z 190,A 39.9052,B 1.149,C -0.008,E1 1.2751,E2 414.3418} C_DIS
LIN {X 102.734,Y 91.4937,Z 190,A 41.5928,B 1.149,C -0.0113,E1 1.272,E2 412.6756} C_DIS
LIN {X 99.7862,Y 94.7002,Z 190,A 43.2551,B 1.149,C -0.0146,E1 1.2689,E2 411.0312} C_DIS
LIN {X 96.6617,Y 97.8874,Z 190,A 44.967,B 1.149,C -0.0179,E1 1.2655,E2 409.3368} C_DIS
LIN {X 93.4334,Y 100.9733,Z 190,A 46.6755,B 1.149,C -0.0211,E1 1.2621,E2 407.6461} C_DIS
LIN {X 90.0237,Y 104.0244,Z 190,A 48.4178,B 1.1488,C -0.0242,E1 1.2584,E2 405.9231} C_DIS
LIN {X 86.7357,Y 106.7816,Z 190,A 50.0423,B 1.1488,C -0.027,E1 1.255,E2 404.3177} C_DIS
LIN {X 83.278,Y 109.4995,Z 190,A 51.7492,B 1.1488,C -0.03,E1 1.2512,E2 402.6255} C_DIS
LIN {X 79.976,Y 111.9334,Z 190,A 53.2579,B 1.1486,C -0.0323,E1 1.2478,E2 401.1402} C_DIS
LIN {X 76.6402,Y 114.2437,Z 190,A 54.8911,B 1.1486,C -0.0351,E1 1.244,E2 399.5138} C_DIS
LIN {X 72.8061,Y 116.7241,Z 190,A 56.6398,B 1.1485,C -0.0378,E1 1.2399,E2 397.783} C_DIS
LIN {X 69.6443,Y 118.6378,Z 190,A 58.1397,B 1.1484,C -0.0402,E1 1.2363,E2 396.2879} C_DIS
LIN {X 65.4096,Y 121.0246,Z 190,A 59.99,B 1.1484,C -0.0428,E1 1.2318,E2 394.4579} C_DIS
LIN {X 61.3847,Y 123.1135,Z 190,A 61.616,B 1.1482,C -0.0447,E1 1.2278,E2 392.8625} C_DIS
LIN {X 58.0458,Y 124.7216,Z 190,A 62.9987,B 1.1482,C -0.0463,E1 1.2244,E2 391.4984} C_DIS
LIN {X 54.7874,Y 126.1867,Z 190,A 64.5428,B 1.1481,C -0.0487,E1 1.2204,E2 389.9481} C_DIS
LIN {X 51.4756,Y 127.5734,Z 190,A 65.7904,B 1.1481,C -0.0498,E1 1.2172,E2 388.7291} C_DIS
LIN {X 47.3665,Y 129.1576,Z 190,A 67.5786,B 1.1479,C -0.052,E1 1.2125,E2 386.9466} C_DIS
LIN {X 43.7745,Y 130.4171,Z 190,A 69.1432,B 1.1479,C -0.0539,E1 1.2084,E2 385.3846} C_DIS
LIN {X 40.2765,Y 131.5391,Z 190,A 70.6299,B 1.1478,C -0.0555,E1 1.2044,E2 383.9032} C_DIS
LIN {X 36.5968,Y 132.6108,Z 190,A 72.2256,B 1.1477,C -0.0573,E1 1.2,E2 382.308} C_DIS
LIN {X 32.5975,Y 133.6499,Z 190,A 73.7716,B 1.1477,C -0.0585,E1 1.1959,E2 380.7823} C_DIS
LIN {X 29.226,Y 134.4271,Z 190,A 75.115,B 1.1476,C -0.0595,E1 1.1922,E2 379.4503} C_DIS
LIN {X 26.2939,Y 135.0319,Z 190,A 76.3355,B 1.1476,C -0.0606,E1 1.1889,E2 378.2331} C_DIS
LIN {X 22.8628,Y 135.6544,Z 190,A 78.2371,B 1.1474,C -0.0632,E1 1.1834,E2 376.281} C_DIS
LIN {X 18.2918,Y 136.3465,Z 190,A 79.4504,B 1.1474,C -0.0624,E1 1.1803,E2 375.149} C_DIS
LIN {X 15.4294,Y 136.7011,Z 190,A 80.9585,B 1.1474,C -0.0642,E1 1.176,E2 373.6067} C_DIS
LIN {X 10.3393,Y 137.1788,Z 190,A 82.6245,B 1.1474,C -0.0642,E1 1.1714,E2 371.9935} C_DIS
LIN {X 7.3321,Y 137.3727,Z 190,A 84.1561,B 1.1472,C -0.0656,E1 1.167,E2 370.4314} C_DIS
LIN {X 2.8227,Y 137.5397,Z 190,A 86.3745,B 1.1472,C -0.0674,E1 1.1607,E2 368.1754} C_DIS
LIN {X -1.6004,Y 137.56,Z 190,A 87.663,B 1.1472,C -0.0666,E1 1.1572,E2 366.95} C_DIS
LIN {X -4.5461,Y 137.4943,Z 190,A 89.4503,B 1.1471,C -0.0684,E1 1.152,E2 365.1002} C_DIS
LIN {X -9.1857,Y 137.2624,Z 190,A 90.9817,B 1.1471,C -0.0678,E1 1.1478,E2 363.6151} C_DIS
LIN {X -13.3621,Y 136.9172,Z 190,A 92.5843,B 1.1471,C -0.0677,E1 1.1434,E2 362.0293} C_DIS
LIN {X -16.2115,Y 136.6089,Z 190,A 94.1333,B 1.1471,C -0.0685,E1 1.1389,E2 360.4409} C_DIS
LIN {X -20.0294,Y 136.1027,Z 190,A 95.5232,B 1.1471,C -0.068,E1 1.1351,E2 359.0758} C_DIS
LIN {X -23.776,Y 135.4979,Z 190,A 96.8981,B 1.1471,C -0.0674,E1 1.1314,E2 357.7247} C_DIS
LIN {X -27.3264,Y 134.826,Z 190,A 98.4753,B 1.1471,C -0.0674,E1 1.127,E2 356.1401} C_DIS
LIN {X -30.1058,Y 134.2337,Z 190,A 99.5348,B 1.1471,C -0.0668,E1 1.1241,E2 355.095} C_DIS
LIN {X -33.7128,Y 133.3724,Z 190,A 101.221,B 1.1471,C -0.0667,E1 1.1194,E2 353.3937} C_DIS
LIN {X -36.677,Y 132.5884,Z 190,A 102.5761,B 1.1471,C -0.0663,E1 1.1157,E2 352.0305} C_DIS
LIN {X -40.1701,Y 131.5716,Z 190,A 104.0435,B 1.1472,C -0.0656,E1 1.1118,E2 350.5692} C_DIS
LIN {X -42.7317,Y 130.7644,Z 190,A 106.1066,B 1.1472,C -0.0666,E1 1.106,E2 348.4} C_DIS
LIN {X -48.7046,Y 128.6577,Z 190,A 108.0663,B 1.1473,C -0.0639,E1 1.101,E2 346.5187} C_DIS
LIN {X -52.1729,Y 127.2923,Z 190,A 110.1544,B 1.1473,C -0.0635,E1 1.0954,E2 344.3709} C_DIS
LIN {X -56.6859,Y 125.3464,Z 190,A 111.7884,B 1.1475,C -0.0613,E1 1.0913,E2 342.7849} C_DIS
LIN {X -60.5454,Y 123.5276,Z 190,A 113.4619,B 1.1475,C -0.0596,E1 1.0871,E2 341.124} C_DIS
LIN {X -63.683,Y 121.9395,Z 190,A 114.9958,B 1.1476,C -0.0583,E1 1.0832,E2 339.5832} C_DIS
LIN {X -67.4911,Y 119.8758,Z 190,A 116.925,B 1.1477,C -0.0566,E1 1.0785,E2 337.6409} C_DIS
LIN {X -70.52,Y 118.1194,Z 190,A 118.4589,B 1.1477,C -0.055,E1 1.0747,E2 336.0993} C_DIS
LIN {X -73.0448,Y 116.5757,Z 190,A 119.9314,B 1.1478,C -0.0538,E1 1.0711,E2 334.6003} C_DIS
LIN {X -77.1196,Y 113.9202,Z 190,A 121.8524,B 1.148,C -0.0512,E1 1.0667,E2 332.6925} C_DIS
LIN {X -82.1835,Y 110.3227,Z 190,A 125.399,B 1.148,C -0.0483,E1 1.0584,E2 329.0373} C_DIS
LIN {X -86.4583,Y 107.0057,Z 190,A 127.056,B 1.1482,C -0.0446,E1 1.0549,E2 327.4505} C_DIS
LIN {X -91.5097,Y 102.7195,Z 190,A 130.3202,B 1.1484,C -0.0405,E1 1.0478,E2 324.1299} C_DIS
LIN {X -95.3934,Y 99.1237,Z 190,A 132.542,B 1.1485,C -0.0367,E1 1.0433,E2 321.9075} C_DIS
LIN {X -98.543,Y 95.9932,Z 190,A 134.2611,B 1.1486,C -0.0334,E1 1.0399,E2 320.2048} C_DIS
LIN {X -102.6078,Y 91.6346,Z 190,A 137.1002,B 1.1487,C -0.0289,E1 1.0344,E2 317.326} C_DIS
LIN {X -105.2001,Y 88.6465,Z 190,A 139.4811,B 1.1488,C -0.0258,E1 1.0299,E2 314.8602} C_DIS
LIN {X -107.9134,Y 85.3237,Z 190,A 140.9028,B 1.1488,C -0.0221,E1 1.0275,E2 313.4827} C_DIS
LIN {X -110.64,Y 81.7568,Z 190,A 143.0912,B 1.149,C -0.0182,E1 1.0238,E2 311.258} C_DIS
LIN {X -113.1339,Y 78.2694,Z 190,A 145.0205,B 1.149,C -0.0144,E1 1.0206,E2 309.3129} C_DIS
LIN {X -115.4903,Y 74.748,Z 190,A 147.0216,B 1.149,C -0.0105,E1 1.0175,E2 307.2849} C_DIS
LIN {X -117.2503,Y 71.9556,Z 190,A 148.8572,B 1.149,C -0.0073,E1 1.0147,E2 305.3952} C_DIS
LIN {X -119.1152,Y 68.8246,Z 190,A 150.213,B 1.149,C -0.0038,E1 1.0128,E2 304.0598} C_DIS
LIN {X -121.484,Y 64.5505,Z 190,A 152.5408,B 1.149,C 0.0011,E1 1.0097,E2 301.6982} C_DIS
LIN {X -123.6998,Y 60.1962,Z 190,A 154.8414,B 1.149,C 0.0061,E1 1.0068,E2 299.3669} C_DIS
LIN {X -125.4806,Y 56.3858,Z 190,A 156.565,B 1.149,C 0.0104,E1 1.0048,E2 297.6478} C_DIS
LIN {X -126.7322,Y 53.5157,Z 190,A 158.0197,B 1.149,C 0.0137,E1 1.0031,E2 296.1757} C_DIS
LIN {X -128.1097,Y 50.1268,Z 190,A 159.8804,B 1.149,C 0.0177,E1 1.0012,E2 294.2749} C_DIS
LIN {X -129.2683,Y 47.0594,Z 190,A 161.4598,B 1.149,C 0.0213,E1 0.9996,E2 292.6703} C_DIS
LIN {X -130.3286,Y 44.0403,Z 190,A 162.8188,B 1.1488,C 0.0248,E1 0.9984,E2 291.309} C_DIS
LIN {X -131.1984,Y 41.3758,Z 190,A 164.2042,B 1.1488,C 0.028,E1 0.9972,E2 289.8974} C_DIS
LIN {X -132.2817,Y 37.7737,Z 190,A 165.983,B 1.1486,C 0.0322,E1 0.9957,E2 288.0936} C_DIS
LIN {X -133.051,Y 34.9631,Z 190,A 167.3591,B 1.1486,C 0.0356,E1 0.9947,E2 286.698} C_DIS
LIN {X -133.6906,Y 32.4287,Z 190,A 168.6177,B 1.1485,C 0.0386,E1 0.9939,E2 285.419} C_DIS
LIN {X -134.631,Y 28.2815,Z 190,A 170.8212,B 1.1483,C 0.0436,E1 0.9925,E2 283.1626} C_DIS
LIN {X -135.3778,Y 24.4474,Z 190,A 172.5374,B 1.1481,C 0.0481,E1 0.9916,E2 281.4361} C_DIS
LIN {X -135.9241,Y 21.2003,Z 190,A 173.9748,B 1.1479,C 0.0519,E1 0.991,E2 279.9912} C_DIS
LIN {X -136.3046,Y 18.6117,Z 190,A 175.4926,B 1.1478,C 0.0552,E1 0.9904,E2 278.4201} C_DIS
LIN {X -136.8011,Y 14.502,Z 190,A 177.356,B 1.1475,C 0.0601,E1 0.9898,E2 276.54} C_DIS
LIN {X -137.1887,Y 10.2037,Z 190,A 179.3721,B 1.1472,C 0.0652,E1 0.9893,E2 274.497} C_DIS
LIN {X -137.4268,Y 6.2552,Z 190,A -178.7598,B 1.147,C 0.0699,E1 0.9891,E2 272.6018} C_DIS
LIN {X -137.5341,Y 3.1162,Z 190,A -177.1224,B 1.1467,C 0.0738,E1 0.9889,E2 270.9228} C_DIS
LIN {X -137.5623,Y -1.3453,Z 190,A -175.0255,B 1.1464,C 0.0791,E1 0.9889,E2 268.796} C_DIS
LIN {X -137.4625,Y -5.3742,Z 190,A -173.1911,B 1.146,C 0.0839,E1 0.9891,E2 266.9424} C_DIS
LIN {X -137.2431,Y -9.458,Z 190,A -171.293,B 1.1457,C 0.0887,E1 0.9894,E2 265.0199} C_DIS
LIN {X -137.0177,Y -12.3085,Z 190,A -169.7556,B 1.1454,C 0.0922,E1 0.9898,E2 263.4379} C_DIS
LIN {X -136.6045,Y -16.2487,Z 190,A -168.0181,B 1.145,C 0.0968,E1 0.9904,E2 261.6897} C_DIS
LIN {X -136.0861,Y -20.1457,Z 190,A -166.0589,B 1.1446,C 0.1015,E1 0.9911,E2 259.689} C_DIS
LIN {X -135.5199,Y -23.6531,Z 190,A -164.5279,B 1.1442,C 0.1056,E1 0.9919,E2 258.152} C_DIS
LIN {X -134.8203,Y -27.3542,Z 190,A -162.7318,B 1.1438,C 0.1099,E1 0.9928,E2 256.3266} C_DIS
LIN {X -134.2276,Y -30.1327,Z 190,A -161.3092,B 1.1435,C 0.1132,E1 0.9937,E2 254.8727} C_DIS
LIN {X -133.3993,Y -33.6069,Z 190,A -159.8704,B 1.1431,C 0.1172,E1 0.9947,E2 253.441} C_DIS
LIN {X -132.5637,Y -36.7651,Z 190,A -158.1046,B 1.1427,C 0.1209,E1 0.996,E2 251.6217} C_DIS
Enddeposition()
END
